KUKA KRL program: MyProgram_183().src

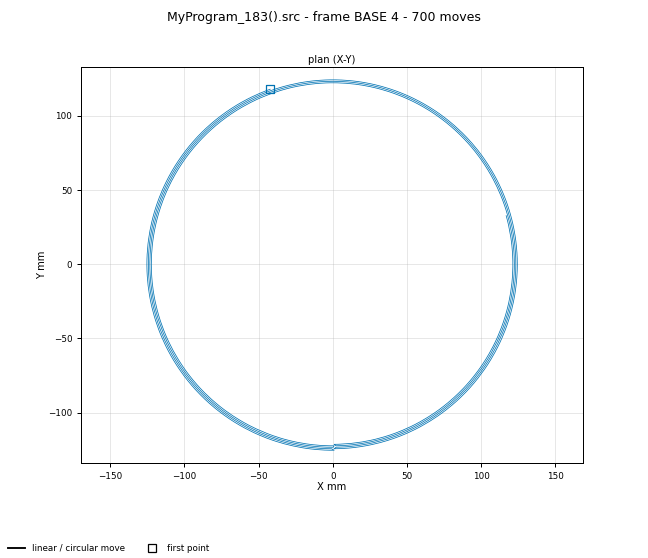
[picture p0: tool path of MyProgram_183().src in frame BASE 4, 700 of 700 moves have a stored position in this frame; points joined in program order, loops and branches not executed]
&ACCESS RVP
&REL 1
&PARAM TEMPLATE = C:\KRC\Roboter\Template\vorgabe
&PARAM EDITMASK = *
DEF MyProgram_183()
; ---- Setting reference (Base) ----
$BASE = BASE_DATA[4]

; --------------------------
; ---- Setting tool (TCP) ----
$TOOL = TOOL_DATA[3]
; --------------------------

$VEL.CP = VEL_APROX_PRINT
Startdeposition()
$VEL.CP = VEL_PRINT
LIN {X -42.2128,Y 118.0054,Z 134,A 105.9576,B 24.9444,C -1.7229,E1 24.9453,E2 340.2664} C_DIS
LIN {X -45.2291,Y 116.8823,Z 134,A 107.4306,B 24.9444,C -1.721,E1 24.9415,E2 338.7949} C_DIS
LIN {X -49.3483,Y 115.2042,Z 134,A 109.5085,B 24.9446,C -1.7201,E1 24.9361,E2 336.7143} C_DIS
LIN {X -52.4065,Y 113.845,Z 134,A 110.9287,B 24.945,C -1.7127,E1 24.9326,E2 335.3083} C_DIS
LIN {X -54.737,Y 112.7456,Z 134,A 112.3481,B 24.9444,C -1.722,E1 24.9289,E2 333.8631} C_DIS
LIN {X -57.7045,Y 111.2549,Z 134,A 113.8311,B 24.9447,C -1.7178,E1 24.9253,E2 332.3861} C_DIS
LIN {X -61.6733,Y 109.1057,Z 134,A 115.8056,B 24.9452,C -1.71,E1 24.9205,E2 330.4243} C_DIS
LIN {X -64.714,Y 107.3297,Z 134,A 117.5198,B 24.9451,C -1.7119,E1 24.9163,E2 328.7004} C_DIS
LIN {X -68.5088,Y 104.9484,Z 134,A 119.5092,B 24.9455,C -1.7052,E1 24.9117,E2 326.7206} C_DIS
LIN {X -71.9101,Y 102.6481,Z 134,A 121.4856,B 24.9455,C -1.706,E1 24.9071,E2 324.7356} C_DIS
LIN {X -75.2001,Y 100.2627,Z 134,A 123.3676,B 24.9456,C -1.7032,E1 24.9029,E2 322.8536} C_DIS
LIN {X -78.7307,Y 97.5142,Z 134,A 125.3322,B 24.9462,C -1.695,E1 24.8986,E2 320.9012} C_DIS
LIN {X -81.914,Y 94.856,Z 134,A 127.2839,B 24.9462,C -1.6933,E1 24.8944,E2 318.9461} C_DIS
LIN {X -85.115,Y 91.9953,Z 134,A 129.2878,B 24.9464,C -1.6905,E1 24.8903,E2 316.9406} C_DIS
LIN {X -88.2175,Y 89.0238,Z 134,A 131.2363,B 24.9468,C -1.6851,E1 24.8864,E2 314.997} C_DIS
LIN {X -91.0515,Y 86.1231,Z 134,A 133.1002,B 24.9471,C -1.6809,E1 24.8828,E2 313.1351} C_DIS
LIN {X -93.789,Y 83.1336,Z 134,A 134.9639,B 24.9473,C -1.6766,E1 24.8793,E2 311.2732} C_DIS
LIN {X -96.7243,Y 79.6996,Z 134,A 137.0122,B 24.9477,C -1.6704,E1 24.8757,E2 309.2303} C_DIS
LIN {X -99.3061,Y 76.4591,Z 134,A 138.9694,B 24.9479,C -1.6681,E1 24.8723,E2 307.2693} C_DIS
LIN {X -101.7154,Y 73.2235,Z 134,A 140.8408,B 24.9481,C -1.6643,E1 24.8692,E2 305.398} C_DIS
LIN {X -104.0135,Y 69.9207,Z 134,A 142.6859,B 24.9484,C -1.6593,E1 24.8663,E2 303.5555} C_DIS
LIN {X -106.3234,Y 66.3544,Z 134,A 144.6,B 24.9488,C -1.6525,E1 24.8634,E2 301.6481} C_DIS
LIN {X -108.4861,Y 62.7559,Z 134,A 146.4839,B 24.9493,C -1.6452,E1 24.8608,E2 299.7716} C_DIS
LIN {X -110.4801,Y 59.1752,Z 134,A 148.3446,B 24.9497,C -1.6391,E1 24.8583,E2 297.9157} C_DIS
LIN {X -112.2559,Y 55.7297,Z 134,A 150.1087,B 24.95,C -1.6334,E1 24.8561,E2 296.1557} C_DIS
LIN {X -113.6473,Y 52.834,Z 134,A 151.5899,B 24.9502,C -1.6295,E1 24.8543,E2 294.6757} C_DIS
LIN {X -114.9101,Y 50.0286,Z 134,A 152.9838,B 24.9505,C -1.6246,E1 24.8527,E2 293.2859} C_DIS
LIN {X -116.1361,Y 47.1124,Z 134,A 154.4266,B 24.9508,C -1.62,E1 24.8512,E2 291.8461} C_DIS
LIN {X -117.0936,Y 44.6855,Z 134,A 155.7763,B 24.9506,C -1.6233,E1 24.8498,E2 290.481} C_DIS
LIN {X -118.3112,Y 41.3481,Z 134,A 157.2703,B 24.9513,C -1.6123,E1 24.8485,E2 289.0046} C_DIS
LIN {X -119.2715,Y 38.4909,Z 134,A 158.6738,B 24.9515,C -1.6091,E1 24.8472,E2 287.6008} C_DIS
LIN {X -120.2509,Y 35.3108,Z 134,A 160.1325,B 24.9519,C -1.6014,E1 24.8461,E2 286.1519} C_DIS
LIN {X -121.2912,Y 31.5618,Z 134,A 162.127,B 24.9517,C -1.6054,E1 24.8446,E2 284.1364} C_DIS
LIN {X -122.0537,Y 28.467,Z 134,A 163.5459,B 24.9521,C -1.5989,E1 24.8437,E2 282.7246} C_DIS
LIN {X -122.7572,Y 25.2565,Z 134,A 164.9795,B 24.9526,C -1.591,E1 24.8429,E2 281.3015} C_DIS
LIN {X -123.2656,Y 22.6512,Z 134,A 166.2569,B 24.9526,C -1.5899,E1 24.8422,E2 280.0191} C_DIS
LIN {X -123.8062,Y 19.4749,Z 134,A 167.6166,B 24.9532,C -1.58,E1 24.8416,E2 278.6749} C_DIS
LIN {X -124.2273,Y 16.5782,Z 134,A 169.0665,B 24.9532,C -1.5806,E1 24.841,E2 277.2148} C_DIS
LIN {X -124.5803,Y 13.6749,Z 134,A 170.3322,B 24.9536,C -1.573,E1 24.8406,E2 275.9597} C_DIS
LIN {X -124.9891,Y 9.2159,Z 134,A 172.3518,B 24.9541,C -1.5651,E1 24.8402,E2 273.9469} C_DIS
LIN {X -125.1413,Y 6.87,Z 134,A 173.5919,B 24.9539,C -1.569,E1 24.84,E2 272.6901} C_DIS
LIN {X -125.2828,Y 3.3838,Z 134,A 175.1553,B 24.9543,C -1.5623,E1 24.8398,E2 271.1331} C_DIS
LIN {X -125.3282,Y -0.6113,Z 134,A 177.0633,B 24.9544,C -1.56,E1 24.8398,E2 269.2192} C_DIS
LIN {X -125.2421,Y -4.6552,Z 134,A 178.83,B 24.955,C -1.5502,E1 24.8399,E2 267.4651} C_DIS
LIN {X -125.0735,Y -7.9936,Z 134,A -179.497,B 24.9549,C -1.5518,E1 24.8402,E2 265.7783} C_DIS
LIN {X -124.7744,Y -11.772,Z 134,A -178.0165,B 24.9559,C -1.5348,E1 24.8406,E2 264.3294} C_DIS
LIN {X -124.4807,Y -14.5538,Z 134,A -176.5766,B 24.9557,C -1.5379,E1 24.841,E2 262.8734} C_DIS
LIN {X -124.086,Y -17.6024,Z 134,A -175.2591,B 24.9562,C -1.5294,E1 24.8415,E2 261.5683} C_DIS
LIN {X -123.6205,Y -20.6188,Z 134,A -173.8852,B 24.9565,C -1.524,E1 24.8421,E2 260.1991} C_DIS
LIN {X -122.8716,Y -24.6945,Z 134,A -171.8482,B 24.9565,C -1.5244,E1 24.8432,E2 258.1492} C_DIS
LIN {X -122.0036,Y -28.6837,Z 134,A -169.8902,B 24.9565,C -1.5226,E1 24.8444,E2 256.1838} C_DIS
LIN {X -121.1814,Y -31.9735,Z 134,A -168.6179,B 24.9576,C -1.5053,E1 24.8452,E2 254.9455} C_DIS
LIN {X -120.4925,Y -34.4857,Z 134,A -167.1064,B 24.9569,C -1.5161,E1 24.8464,E2 253.3995} C_DIS
LIN {X -119.479,Y -37.8414,Z 134,A -165.6096,B 24.9575,C -1.5064,E1 24.8476,E2 251.9173} C_DIS
LIN {X -118.4872,Y -40.8404,Z 134,A -164.2077,B 24.9578,C -1.5001,E1 24.8489,E2 250.5223} C_DIS
LIN {X -117.4756,Y -43.6657,Z 134,A -162.801,B 24.958,C -1.4975,E1 24.8502,E2 249.1137} C_DIS
LIN {X -116.5014,Y -46.2062,Z 134,A -161.5799,B 24.9583,C -1.4928,E1 24.8515,E2 247.8971} C_DIS
LIN {X -115.2168,Y -49.3193,Z 134,A -159.9549,B 24.9583,C -1.4922,E1 24.8532,E2 246.2646} C_DIS
LIN {X -113.8491,Y -52.3977,Z 134,A -158.5355,B 24.9588,C -1.4822,E1 24.8549,E2 244.8611} C_DIS
LIN {X -112.7456,Y -54.737,Z 134,A -157.1048,B 24.9584,C -1.4901,E1 24.8566,E2 243.4038} C_DIS
LIN {X -111.2809,Y -57.6551,Z 134,A -155.6229,B 24.9587,C -1.4854,E1 24.8585,E2 241.9251} C_DIS
LIN {X -109.093,Y -61.6959,Z 134,A -153.6286,B 24.9593,C -1.4748,E1 24.8612,E2 239.9458} C_DIS
LIN {X -107.3297,Y -64.714,Z 134,A -151.9247,B 24.9593,C -1.4753,E1 24.8636,E2 238.2318} C_DIS
LIN {X -104.937,Y -68.5264,Z 134,A -149.9496,B 24.9597,C -1.466,E1 24.8666,E2 236.2688} C_DIS
LIN {X -102.7847,Y -71.7138,Z 134,A -148.1115,B 24.9597,C -1.4652,E1 24.8695,E2 234.4236} C_DIS
LIN {X -100.283,Y -75.1732,Z 134,A -146.0743,B 24.9598,C -1.4642,E1 24.8729,E2 232.3788} C_DIS
LIN {X -97.8084,Y -78.3659,Z 134,A -144.28,B 24.9602,C -1.4573,E1 24.876,E2 230.5925} C_DIS
LIN {X -95.2021,Y -81.5121,Z 134,A -142.348,B 24.9602,C -1.4559,E1 24.8795,E2 228.655} C_DIS
LIN {X -92.3809,Y -84.6955,Z 134,A -140.4316,B 24.9606,C -1.4501,E1 24.883,E2 226.7438} C_DIS
LIN {X -89.3624,Y -87.8744,Z 134,A -138.4231,B 24.9608,C -1.4459,E1 24.8869,E2 224.7366} C_DIS
LIN {X -86.2984,Y -90.8861,Z 134,A -136.419,B 24.961,C -1.4436,E1 24.891,E2 222.7298} C_DIS
LIN {X -83.1336,Y -93.789,Z 134,A -134.4735,B 24.9612,C -1.4388,E1 24.895,E2 220.7879} C_DIS
LIN {X -79.7295,Y -96.6996,Z 134,A -132.4395,B 24.9615,C -1.4342,E1 24.8993,E2 218.757} C_DIS
LIN {X -76.4591,Y -99.3061,Z 134,A -130.4738,B 24.9615,C -1.4332,E1 24.9037,E2 216.7865} C_DIS
LIN {X -73.119,Y -101.7901,Z 134,A -128.5626,B 24.9617,C -1.4303,E1 24.908,E2 214.8755} C_DIS
LIN {X -69.4511,Y -104.327,Z 134,A -126.6149,B 24.9621,C -1.4226,E1 24.9124,E2 212.9395} C_DIS
LIN {X -66.3544,Y -106.3234,Z 134,A -124.8572,B 24.9621,C -1.4235,E1 24.9166,E2 211.1743} C_DIS
LIN {X -62.6309,Y -108.5585,Z 134,A -122.9402,B 24.9624,C -1.4173,E1 24.9212,E2 209.266} C_DIS
LIN {X -59.1752,Y -110.4801,Z 134,A -121.0908,B 24.9624,C -1.4168,E1 24.9257,E2 207.4125} C_DIS
LIN {X -55.7324,Y -112.2545,Z 134,A -119.3679,B 24.9626,C -1.4123,E1 24.93,E2 205.6957} C_DIS
LIN {X -53.315,Y -113.4249,Z 134,A -118.0043,B 24.9624,C -1.4173,E1 24.9335,E2 204.317} C_DIS
LIN {X -50.0286,Y -114.9101,Z 134,A -116.5037,B 24.9628,C -1.4084,E1 24.9373,E2 202.8339} C_DIS
LIN {X -47.0776,Y -116.1501,Z 134,A -115.0402,B 24.9629,C -1.4069,E1 24.9411,E2 201.3706} C_DIS
LIN {X -44.6855,Y -117.0936,Z 134,A -113.712,B 24.9626,C -1.413,E1 24.9446,E2 200.025} C_DIS
LIN {X -41.3481,Y -118.3112,Z 134,A -112.237,B 24.9631,C -1.4044,E1 24.9484,E2 198.5675} C_DIS
LIN {X -38.3419,Y -119.3191,Z 134,A -110.8033,B 24.9631,C -1.4025,E1 24.9522,E2 197.1356} C_DIS
LIN {X -35.3348,Y -120.2439,Z 134,A -109.3676,B 24.9632,C -1.4014,E1 24.956,E2 195.7002} C_DIS
LIN {X -32.5893,Y -121.0172,Z 134,A -108.2282,B 24.9637,C -1.3926,E1 24.9591,E2 194.58} C_DIS
LIN {X -29.5959,Y -121.7837,Z 134,A -106.7428,B 24.9635,C -1.3953,E1 24.9631,E2 193.086} C_DIS
LIN {X -26.6178,Y -122.469,Z 134,A -105.2134,B 24.9632,C -1.401,E1 24.9673,E2 191.5412} C_DIS
LIN {X -23.8287,Y -123.0424,Z 134,A -104.0673,B 24.9637,C -1.3929,E1 24.9704,E2 190.413} C_DIS
LIN {X -20.9206,Y -123.5701,Z 134,A -102.555,B 24.9633,C -1.4002,E1 24.9746,E2 188.8816} C_DIS
LIN {X -18.2655,Y -123.9913,Z 134,A -101.2825,B 24.9632,C -1.402,E1 24.9781,E2 187.6039} C_DIS
LIN {X -14.8953,Y -124.44,Z 134,A -99.7709,B 24.9633,C -1.3997,E1 24.9823,E2 186.0967} C_DIS
LIN {X -11.2615,Y -124.8234,Z 134,A -97.9671,B 24.963,C -1.406,E1 24.9874,E2 184.2769} C_DIS
LIN {X -7.9927,Y -125.0736,Z 134,A -96.7028,B 24.9636,C -1.3946,E1 24.9908,E2 183.0393} C_DIS
LIN {X -5.5873,Y -125.2058,Z 134,A -95.4107,B 24.9631,C -1.404,E1 24.9945,E2 181.7246} C_DIS
LIN {X -2.2482,Y -125.3084,Z 134,A -94.08,B 24.9636,C -1.3946,E1 24.9981,E2 180.416} C_DIS
LIN {X 0.8896,Y -125.3254,Z 134,A -92.9496,B 24.9643,C -1.38,E1 25.0012,E2 179.3201} C_DIS
Enddeposition()
LIN {X 0.8896,Y -125.3254,Z 134,A -92.9496,B 24.9643,C -1.38,E1 25.0012,E2 179.3201} C_DIS
Startdeposition()
$VEL.CP = VEL_PRINT
LIN {X -0.8291,Y -124.3295,Z 134,A -94.093,B 24.9643,C -1.3803,E1 24.998,E2 180.4627} C_DIS
LIN {X -4.7488,Y -124.2414,Z 134,A -95.8527,B 24.9643,C -1.3824,E1 24.9931,E2 182.2179} C_DIS
LIN {X -8.5607,Y -124.038,Z 134,A -97.7312,B 24.9645,C -1.3766,E1 24.9878,E2 184.1107} C_DIS
LIN {X -13.0048,Y -123.6503,Z 134,A -99.6905,B 24.9643,C -1.3814,E1 24.9824,E2 186.0598} C_DIS
LIN {X -16.1934,Y -123.2729,Z 134,A -101.1295,B 24.9641,C -1.3836,E1 24.9784,E2 187.4945} C_DIS
LIN {X -19.8425,Y -122.7399,Z 134,A -102.89,B 24.9643,C -1.3811,E1 24.9736,E2 189.2625} C_DIS
LIN {X -24.0406,Y -121.9876,Z 134,A -104.8827,B 24.9643,C -1.3805,E1 24.9681,E2 191.2585} C_DIS
LIN {X -27.1247,Y -121.3383,Z 134,A -106.231,B 24.964,C -1.3861,E1 24.9644,E2 192.5951} C_DIS
LIN {X -30.2211,Y -120.6036,Z 134,A -107.7557,B 24.9641,C -1.3842,E1 24.9603,E2 194.1265} C_DIS
LIN {X -34.3893,Y -119.4825,Z 134,A -109.7988,B 24.9641,C -1.383,E1 24.9548,E2 196.1758} C_DIS
LIN {X -41.2804,Y -117.2802,Z 134,A -113.1988,B 24.9641,C -1.3825,E1 24.9457,E2 199.5831} C_DIS
LIN {X -44.9084,Y -115.938,Z 134,A -114.9299,B 24.964,C -1.3867,E1 24.9412,E2 201.308} C_DIS
LIN {X -48.9847,Y -114.276,Z 134,A -117.101,B 24.9642,C -1.3822,E1 24.9356,E2 203.4948} C_DIS
LIN {X -53.007,Y -112.4679,Z 134,A -119.021,B 24.9638,C -1.3897,E1 24.9308,E2 205.4016} C_DIS
LIN {X -55.7905,Y -111.1136,Z 134,A -120.4058,B 24.9636,C -1.3934,E1 24.9273,E2 206.7812} C_DIS
LIN {X -58.7245,Y -109.5913,Z 134,A -121.9414,B 24.9636,C -1.3949,E1 24.9235,E2 208.3176} C_DIS
LIN {X -62.3051,Y -107.5959,Z 134,A -123.8517,B 24.9635,C -1.3966,E1 24.9189,E2 210.2295} C_DIS
LIN {X -66.3823,Y -105.1294,Z 134,A -126.041,B 24.9633,C -1.4002,E1 24.9137,E2 212.417} C_DIS
LIN {X -69.9315,Y -102.803,Z 134,A -128.0254,B 24.9632,C -1.4021,E1 24.9091,E2 214.4035} C_DIS
LIN {X -73.3696,Y -100.3782,Z 134,A -129.6623,B 24.9623,C -1.4193,E1 24.9054,E2 216.0052} C_DIS
LIN {X -75.9762,Y -98.4199,Z 134,A -131.4708,B 24.9629,C -1.408,E1 24.9013,E2 217.8471} C_DIS
LIN {X -79.2164,Y -95.8309,Z 134,A -133.4121,B 24.9627,C -1.4102,E1 24.8971,E2 219.7905} C_DIS
LIN {X -82.6197,Y -92.9134,Z 134,A -135.2958,B 24.9621,C -1.4226,E1 24.8932,E2 221.6521} C_DIS
LIN {X -85.1856,Y -90.5662,Z 134,A -137.0947,B 24.9624,C -1.417,E1 24.8895,E2 223.4716} C_DIS
LIN {X -88.264,Y -87.5686,Z 134,A -139.0924,B 24.9622,C -1.4204,E1 24.8855,E2 225.4696} C_DIS
LIN {X -91.3259,Y -84.371,Z 134,A -141.1608,B 24.962,C -1.4237,E1 24.8815,E2 227.5392} C_DIS
LIN {X -93.89,Y -81.5081,Z 134,A -142.9209,B 24.9618,C -1.4283,E1 24.8783,E2 229.2963} C_DIS
LIN {X -96.738,Y -78.106,Z 134,A -144.9464,B 24.9615,C -1.434,E1 24.8747,E2 231.3174} C_DIS
LIN {X -99.4141,Y -74.6707,Z 134,A -146.9963,B 24.9613,C -1.437,E1 24.8712,E2 233.37} C_DIS
LIN {X -101.9099,Y -71.2267,Z 134,A -148.9684,B 24.9611,C -1.4415,E1 24.868,E2 235.3412} C_DIS
LIN {X -103.9347,Y -68.2379,Z 134,A -150.697,B 24.961,C -1.4429,E1 24.8653,E2 237.075} C_DIS
LIN {X -106.3933,Y -64.3372,Z 134,A -152.7469,B 24.9605,C -1.4519,E1 24.8624,E2 239.1139} C_DIS
LIN {X -108.4732,Y -60.7651,Z 134,A -154.8338,B 24.9607,C -1.449,E1 24.8594,E2 241.2186} C_DIS
LIN {X -110.6976,Y -56.6076,Z 134,A -156.8123,B 24.9599,C -1.4638,E1 24.8569,E2 243.1725} C_DIS
LIN {X -112.4921,Y -52.9564,Z 134,A -158.9864,B 24.9603,C -1.4558,E1 24.8543,E2 245.3772} C_DIS
LIN {X -113.8392,Y -49.995,Z 134,A -160.2929,B 24.9596,C -1.4687,E1 24.8528,E2 246.6603} C_DIS
LIN {X -115.3156,Y -46.483,Z 134,A -161.9287,B 24.959,C -1.4792,E1 24.8511,E2 248.2801} C_DIS
LIN {X -116.7566,Y -42.739,Z 134,A -164.3001,B 24.96,C -1.4617,E1 24.8487,E2 250.7067} C_DIS
LIN {X -118.0857,Y -38.9141,Z 134,A -165.7588,B 24.9587,C -1.4853,E1 24.8475,E2 252.1175} C_DIS
LIN {X -119.2653,Y -35.1314,Z 134,A -167.3661,B 24.9578,C -1.5006,E1 24.8462,E2 253.6976} C_DIS
LIN {X -120.1074,Y -32.1344,Z 134,A -168.9132,B 24.9578,C -1.5001,E1 24.845,E2 255.255} C_DIS
LIN {X -120.8429,Y -29.2475,Z 134,A -170.3453,B 24.9578,C -1.5017,E1 24.8441,E2 256.6915} C_DIS
LIN {X -121.6967,Y -25.4715,Z 134,A -173.356,B 24.9604,C -1.4539,E1 24.8423,E2 259.8339} C_DIS
LIN {X -123.0108,Y -18.0842,Z 134,A -175.4738,B 24.9565,C -1.5233,E1 24.8414,E2 261.799} C_DIS
LIN {X -123.6979,Y -12.5594,Z 134,A -178.3129,B 24.9567,C -1.5195,E1 24.8405,E2 264.6641} C_DIS
LIN {X -124.1612,Y -6.522,Z 134,A 178.9873,B 24.956,C -1.5325,E1 24.84,E2 267.349} C_DIS
LIN {X -124.2881,Y -3.3114,Z 134,A 177.0622,B 24.9568,C -1.518,E1 24.8398,E2 269.3205} C_DIS
LIN {X -124.3322,Y 0.5419,Z 134,A 175.6181,B 24.9557,C -1.5382,E1 24.8398,E2 270.725} C_DIS
LIN {X -124.184,Y 6.0687,Z 134,A 173.0923,B 24.9551,C -1.5476,E1 24.84,E2 273.2436} C_DIS
LIN {X -123.9381,Y 9.9053,Z 134,A 171.2479,B 24.955,C -1.5502,E1 24.8404,E2 275.0929} C_DIS
LIN {X -123.5359,Y 14.0627,Z 134,A 169.433,B 24.9543,C -1.5613,E1 24.8409,E2 276.8922} C_DIS
LIN {X -123.093,Y 17.5083,Z 134,A 167.7056,B 24.9543,C -1.561,E1 24.8416,E2 278.6306} C_DIS
LIN {X -122.5787,Y 20.809,Z 134,A 165.4846,B 24.9558,C -1.5364,E1 24.8427,E2 280.9235} C_DIS
LIN {X -121.5645,Y 26.0864,Z 134,A 163.7741,B 24.9534,C -1.5778,E1 24.8436,E2 282.5454} C_DIS
LIN {X -120.8639,Y 29.1601,Z 134,A 162.3759,B 24.9529,C -1.5849,E1 24.8445,E2 283.935} C_DIS
LIN {X -120.0864,Y 32.2132,Z 134,A 160.7926,B 24.953,C -1.5838,E1 24.8456,E2 285.5301} C_DIS
LIN {X -118.9565,Y 36.1635,Z 134,A 158.9999,B 24.9524,C -1.5942,E1 24.847,E2 287.3082} C_DIS
LIN {X -117.9617,Y 39.2863,Z 134,A 157.4009,B 24.9524,C -1.5951,E1 24.8484,E2 288.9142} C_DIS
LIN {X -116.6741,Y 42.965,Z 134,A 155.6314,B 24.9519,C -1.6019,E1 24.85,E2 290.6775} C_DIS
LIN {X -115.3326,Y 46.4408,Z 134,A 153.9134,B 24.9516,C -1.6073,E1 24.8518,E2 292.3924} C_DIS
LIN {X -114.2119,Y 49.133,Z 134,A 152.5,B 24.9516,C -1.6084,E1 24.8533,E2 293.8111} C_DIS
LIN {X -112.8301,Y 52.2275,Z 134,A 151.0165,B 24.951,C -1.6166,E1 24.855,E2 295.283} C_DIS
LIN {X -111.1514,Y 55.7163,Z 134,A 149.0903,B 24.951,C -1.6157,E1 24.8574,E2 297.2217} C_DIS
LIN {X -109.5282,Y 58.842,Z 134,A 147.4976,B 24.9507,C -1.6219,E1 24.8595,E2 298.8081} C_DIS
LIN {X -107.5727,Y 62.3452,Z 134,A 145.6296,B 24.9504,C -1.6265,E1 24.862,E2 300.6749} C_DIS
LIN {X -105.3698,Y 66.001,Z 134,A 143.5621,B 24.9504,C -1.6278,E1 24.8651,E2 302.75} C_DIS
LIN {X -102.9906,Y 69.6545,Z 134,A 141.5508,B 24.95,C -1.6334,E1 24.8682,E2 304.758} C_DIS
LIN {X -100.4113,Y 73.3246,Z 134,A 139.4495,B 24.9497,C -1.6377,E1 24.8716,E2 306.8594} C_DIS
LIN {X -97.72,Y 76.874,Z 134,A 137.431,B 24.9493,C -1.6447,E1 24.875,E2 308.8707} C_DIS
LIN {X -94.9868,Y 80.2276,Z 134,A 135.3766,B 24.9491,C -1.6473,E1 24.8787,E2 310.9284} C_DIS
LIN {X -92.0924,Y 83.5332,Z 134,A 133.4305,B 24.9486,C -1.6561,E1 24.8823,E2 312.8624} C_DIS
LIN {X -89.2646,Y 86.5484,Z 134,A 131.4611,B 24.9485,C -1.658,E1 24.8861,E2 314.8358} C_DIS
LIN {X -86.162,Y 89.6383,Z 134,A 129.4066,B 24.9483,C -1.6612,E1 24.8902,E2 316.8911} C_DIS
LIN {X -83.1514,Y 92.4376,Z 134,A 127.519,B 24.948,C -1.666,E1 24.8941,E2 318.775} C_DIS
LIN {X -79.9464,Y 95.2227,Z 134,A 125.6039,B 24.9476,C -1.6723,E1 24.8981,E2 320.6824} C_DIS
LIN {X -76.572,Y 97.9572,Z 134,A 123.5711,B 24.9474,C -1.6753,E1 24.9026,E2 322.7157} C_DIS
LIN {X -73.3404,Y 100.3997,Z 134,A 121.695,B 24.9472,C -1.6788,E1 24.9068,E2 324.5901} C_DIS
LIN {X -70.114,Y 102.6787,Z 134,A 119.8614,B 24.947,C -1.6819,E1 24.911,E2 326.4226} C_DIS
LIN {X -66.6424,Y 104.9653,Z 134,A 117.9034,B 24.9469,C -1.6838,E1 24.9156,E2 328.3826} C_DIS
LIN {X -62.7596,Y 107.3317,Z 134,A 115.8441,B 24.9465,C -1.6893,E1 24.9205,E2 330.4351} C_DIS
LIN {X -59.0643,Y 109.4088,Z 134,A 113.8454,B 24.9465,C -1.6907,E1 24.9254,E2 332.4362} C_DIS
LIN {X -55.2264,Y 111.3932,Z 134,A 112.2081,B 24.9452,C -1.7101,E1 24.9293,E2 334.0319} C_DIS
LIN {X -51.4492,Y 113.1896,Z 134,A 109.8903,B 24.9461,C -1.6953,E1 24.9353,E2 336.3906} C_DIS
LIN {X -48.0206,Y 114.6839,Z 134,A 108.2868,B 24.9456,C -1.7033,E1 24.9394,E2 337.9787} C_DIS
LIN {X -45.2872,Y 115.7908,Z 134,A 106.3065,B 24.9473,C -1.677,E1 24.9447,E2 340.0259} C_DIS
LIN {X -40.8805,Y 117.4189,Z 134,A 104.7604,B 24.9453,C -1.7079,E1 24.9486,E2 341.5017} C_DIS
LIN {X -37.7579,Y 118.4598,Z 134,A 103.1894,B 24.9453,C -1.7072,E1 24.9528,E2 343.0771} C_DIS
LIN {X -33.5588,Y 119.7172,Z 134,A 100.6802,B 24.9467,C -1.687,E1 24.9597,E2 345.6382} C_DIS
LIN {X -29.4074,Y 120.8043,Z 134,A 99.4701,B 24.9443,C -1.7242,E1 24.9627,E2 346.7617} C_DIS
LIN {X -22.7276,Y 122.2386,Z 134,A 96.0433,B 24.9449,C -1.714,E1 24.9722,E2 350.217} C_DIS
LIN {X -20.3015,Y 122.6634,Z 134,A 94.6081,B 24.9458,C -1.7009,E1 24.9762,E2 351.6844} C_DIS
LIN {X -16.898,Y 123.1803,Z 134,A 93.2781,B 24.945,C -1.7138,E1 24.9798,E2 352.985} C_DIS
LIN {X -13.0642,Y 123.644,Z 134,A 91.5095,B 24.9449,C -1.7153,E1 24.9847,E2 354.751} C_DIS
LIN {X -9.0218,Y 124.0043,Z 134,A 89.6198,B 24.9449,C -1.7153,E1 24.9899,E2 356.6416} C_DIS
LIN {X -5.171,Y 124.2249,Z 134,A 87.9265,B 24.9446,C -1.7199,E1 24.9946,E2 358.3246} C_DIS
LIN {X -1.7803,Y 124.3197,Z 134,A 86.3238,B 24.9446,C -1.7184,E1 24.9991,E2 359.9309} C_DIS
LIN {X 1.8786,Y 124.3181,Z 134,A 84.5937,B 24.9448,C -1.7166,E1 25.004,E2 361.6651} C_DIS
LIN {X 5.9235,Y 124.1913,Z 134,A 82.6719,B 24.9449,C -1.7141,E1 25.0093,E2 363.5923} C_DIS
LIN {X 10.0163,Y 123.9287,Z 134,A 80.9026,B 24.9446,C -1.7197,E1 25.0142,E2 365.3476} C_DIS
LIN {X 13.2988,Y 123.6187,Z 134,A 79.3791,B 24.9446,C -1.7193,E1 25.0185,E2 366.8709} C_DIS
LIN {X 16.8352,Y 123.1888,Z 134,A 77.8073,B 24.9444,C -1.7222,E1 25.0228,E2 368.4346} C_DIS
LIN {X 20.7641,Y 122.5862,Z 134,A 75.8052,B 24.945,C -1.7136,E1 25.0284,E2 370.4553} C_DIS
LIN {X 24.909,Y 121.8112,Z 134,A 73.9642,B 24.9447,C -1.7176,E1 25.0334,E2 372.2845} C_DIS
LIN {X 28.1891,Y 121.0952,Z 134,A 72.2621,B 24.9452,C -1.7094,E1 25.0381,E2 374.0038} C_DIS
LIN {X 32.8459,Y 119.9166,Z 134,A 70.304,B 24.9445,C -1.7202,E1 25.0433,E2 375.9333} C_DIS
LIN {X 38.4183,Y 118.2488,Z 134,A 67.4575,B 24.9452,C -1.7101,E1 25.0509,E2 378.7985} C_DIS
LIN {X 42.0457,Y 117.0066,Z 134,A 65.7953,B 24.945,C -1.7136,E1 25.0553,E2 380.4491} C_DIS
LIN {X 44.879,Y 115.9494,Z 134,A 64.5599,B 24.9446,C -1.7199,E1 25.0584,E2 381.667} C_DIS
LIN {X 48.497,Y 114.4849,Z 134,A 62.5282,B 24.9454,C -1.7066,E1 25.0638,E2 383.7253} C_DIS
LIN {X 51.4448,Y 113.1916,Z 134,A 61.0841,B 24.9454,C -1.7068,E1 25.0674,E2 385.1654} C_DIS
LIN {X 54.3981,Y 111.8018,Z 134,A 59.4753,B 24.9458,C -1.6999,E1 25.0715,E2 386.7864} C_DIS
LIN {X 58.6019,Y 109.6572,Z 134,A 57.3728,B 24.9458,C -1.7005,E1 25.0767,E2 388.8817} C_DIS
LIN {X 61.5153,Y 108.0494,Z 134,A 55.8274,B 24.946,C -1.6977,E1 25.0805,E2 390.429} C_DIS
LIN {X 65.3025,Y 105.8041,Z 134,A 53.8059,B 24.9462,C -1.6949,E1 25.0853,E2 392.4507} C_DIS
LIN {X 68.8681,Y 103.5182,Z 134,A 51.876,B 24.9462,C -1.6929,E1 25.0898,E2 394.3792} C_DIS
LIN {X 71.727,Y 101.5581,Z 134,A 50.2654,B 24.9465,C -1.6895,E1 25.0935,E2 395.9922} C_DIS
LIN {X 75.2073,Y 99.0092,Z 134,A 48.3095,B 24.9466,C -1.6875,E1 25.0979,E2 397.9459} C_DIS
LIN {X 78.4367,Y 96.4706,Z 134,A 46.239,B 24.9474,C -1.6751,E1 25.1024,E2 400.0378} C_DIS
LIN {X 81.8563,Y 93.5861,Z 134,A 43.2776,B 24.9504,C -1.6271,E1 25.1089,E2 403.1009} C_DIS
LIN {X 87.2524,Y 88.577,Z 134,A 40.9535,B 24.9476,C -1.6722,E1 25.1133,E2 405.3089} C_DIS
LIN {X 90.2407,Y 85.5307,Z 134,A 39.0371,B 24.9477,C -1.6703,E1 25.117,E2 407.2215} C_DIS
LIN {X 93.8684,Y 81.5328,Z 134,A 35.6978,B 24.9507,C -1.6225,E1 25.1233,E2 410.6587} C_DIS
LIN {X 97.8335,Y 76.7294,Z 134,A 33.7029,B 24.9484,C -1.6588,E1 25.1267,E2 412.5586} C_DIS
LIN {X 100.4155,Y 73.3188,Z 134,A 32.0034,B 24.9479,C -1.6674,E1 25.1294,E2 414.2295} C_DIS
LIN {X 102.1863,Y 70.8295,Z 134,A 30.3373,B 24.9489,C -1.6509,E1 25.1322,E2 415.9265} C_DIS
LIN {X 104.5096,Y 67.355,Z 134,A 28.3744,B 24.9494,C -1.6439,E1 25.1352,E2 417.8959} C_DIS
LIN {X 106.8778,Y 63.5292,Z 134,A 26.3523,B 24.9495,C -1.6409,E1 25.1381,E2 419.9149} C_DIS
LIN {X 109.0073,Y 59.8022,Z 134,A 24.5598,B 24.9493,C -1.6448,E1 25.1405,E2 421.6888} C_DIS
LIN {X 110.6401,Y 56.7207,Z 134,A 22.9832,B 24.9495,C -1.6419,E1 25.1426,E2 423.264} C_DIS
LIN {X 112.0561,Y 53.8689,Z 134,A 21.3973,B 24.9501,C -1.6317,E1 25.1445,E2 424.8655} C_DIS
LIN {X 113.5493,Y 50.6452,Z 134,A 19.76,B 24.9504,C -1.6269,E1 25.1464,E2 426.5051} C_DIS
LIN {X 114.9681,Y 47.34,Z 134,A 18.0406,B 24.9509,C -1.6189,E1 25.1483,E2 428.234} C_DIS
LIN {X 116.3029,Y 43.9561,Z 134,A 16.4624,B 24.9509,C -1.6189,E1 25.1499,E2 429.8035} C_DIS
LIN {X 117.4019,Y 40.9294,Z 134,A 14.9876,B 24.9511,C -1.6149,E1 25.1513,E2 431.2795} C_DIS
LIN {X 118.6726,Y 37.0909,Z 134,A 12.7365,B 24.9527,C -1.5895,E1 25.1532,E2 433.5777} C_DIS
LIN {X 119.6887,Y 33.6607,Z 134,A 11.4992,B 24.9517,C -1.6052,E1 25.1541,E2 434.7707} C_DIS
LIN {X 120.6461,Y 30.0536,Z 134,A 9.6892,B 24.9523,C -1.5953,E1 25.1554,E2 436.5938} C_DIS
LIN {X 121.32,Y 27.205,Z 134,A 8.2489,B 24.9528,C -1.5864,E1 25.1563,E2 438.0467} C_DIS
LIN {X 122.0732,Y 23.5927,Z 134,A 6.6098,B 24.953,C -1.5841,E1 25.1572,E2 439.6816} C_DIS
LIN {X 122.8174,Y 19.35,Z 134,A 4.7647,B 24.953,C -1.5848,E1 25.158,E2 441.5142} C_DIS
LIN {X 123.3382,Y 15.695,Z 134,A 3.1294,B 24.953,C -1.5827,E1 25.1586,E2 443.1449} C_DIS
LIN {X 123.7731,Y 11.7765,Z 134,A 1.2177,B 24.9537,C -1.572,E1 25.1592,E2 445.0705} C_DIS
LIN {X 124.0952,Y 7.6714,Z 134,A -0.5805,B 24.9537,C -1.5709,E1 25.1595,E2 446.8606} C_DIS
LIN {X 124.2634,Y 4.1838,Z 134,A -2.3622,B 24.9546,C -1.5568,E1 25.1597,E2 448.6649} C_DIS
LIN {X 124.3326,Y -0.4646,Z 134,A -4.3597,B 24.9546,C -1.5571,E1 25.1597,E2 450.6497} C_DIS
LIN {X 124.2505,Y -4.5163,Z 134,A -6.2337,B 24.9549,C -1.5507,E1 25.1597,E2 452.5278} C_DIS
LIN {X 124.0221,Y -8.7778,Z 134,A -8.1363,B 24.9551,C -1.5475,E1 25.1593,E2 454.4266} C_DIS
LIN {X 123.6914,Y -12.6229,Z 134,A -10.1576,B 24.9562,C -1.5292,E1 25.1588,E2 456.479} C_DIS
LIN {X 123.1034,Y -17.4361,Z 134,A -12.1141,B 24.9558,C -1.5361,E1 25.1581,E2 458.4078} C_DIS
LIN {X 122.5568,Y -20.9404,Z 134,A -13.699,B 24.956,C -1.5333,E1 25.1573,E2 459.99} C_DIS
LIN {X 121.7403,Y -25.2573,Z 134,A -15.8465,B 24.9567,C -1.5204,E1 25.1562,E2 462.1554} C_DIS
LIN {X 120.5423,Y -30.4627,Z 134,A -18.1622,B 24.9567,C -1.5198,E1 25.1547,E2 464.4589} C_DIS
LIN {X 119.5443,Y -34.1771,Z 134,A -20.035,B 24.9573,C -1.509,E1 25.1533,E2 466.3465} C_DIS
LIN {X 118.4673,Y -37.7343,Z 134,A -22.1037,B 24.9587,C -1.4854,E1 25.1515,E2 468.459} C_DIS
LIN {X 117.1683,Y -41.5973,Z 134,A -23.5676,B 24.9578,C -1.5005,E1 25.1502,E2 469.8792} C_DIS
LIN {X 116.029,Y -44.6742,Z 134,A -25.0458,B 24.958,C -1.4975,E1 25.1487,E2 471.3562} C_DIS
LIN {X 114.1384,Y -49.303,Z 134,A -27.3023,B 24.9583,C -1.4927,E1 25.1463,E2 473.6115} C_DIS
LIN {X 112.6911,Y -52.5282,Z 134,A -29.0277,B 24.9588,C -1.4828,E1 25.1443,E2 475.3509} C_DIS
LIN {X 110.9836,Y -56.046,Z 134,A -30.6424,B 24.9586,C -1.4868,E1 25.1423,E2 476.9475} C_DIS
LIN {X 109.2985,Y -59.2683,Z 134,A -32.6734,B 24.9599,C -1.4637,E1 25.1396,E2 479.0224} C_DIS
LIN {X 106.5966,Y -64.0009,Z 134,A -34.9749,B 24.9597,C -1.467,E1 25.1364,E2 481.3043} C_DIS
LIN {X 104.3155,Y -67.6541,Z 134,A -36.8626,B 24.9597,C -1.4662,E1 25.1335,E2 483.1844} C_DIS
LIN {X 102.073,Y -70.9923,Z 134,A -38.7466,B 24.9601,C -1.4593,E1 25.1306,E2 485.0752} C_DIS
LIN {X 97.8398,Y -76.7215,Z 134,A -41.9982,B 24.9605,C -1.4518,E1 25.1251,E2 488.329} C_DIS
LIN {X 95.2544,Y -79.9087,Z 134,A -43.8935,B 24.9608,C -1.4466,E1 25.1217,E2 490.2279} C_DIS
LIN {X 92.4664,Y -83.1192,Z 134,A -45.5836,B 24.9603,C -1.4551,E1 25.1187,E2 491.8903} C_DIS
LIN {X 89.3547,Y -86.4554,Z 134,A -48.0777,B 24.9617,C -1.4299,E1 25.1138,E2 494.433} C_DIS
LIN {X 85.8133,Y -89.9716,Z 134,A -50.1803,B 24.9615,C -1.4342,E1 25.1096,E2 496.5167} C_DIS
LIN {X 82.7989,Y -92.7533,Z 134,A -51.8323,B 24.9611,C -1.4417,E1 25.1063,E2 498.1443} C_DIS
LIN {X 80.5677,Y -94.6976,Z 134,A -53.6518,B 24.9625,C -1.4156,E1 25.1023,E2 500.0182} C_DIS
LIN {X 76.4712,Y -98.0362,Z 134,A -55.929,B 24.9623,C -1.4181,E1 25.0974,E2 502.2811} C_DIS
LIN {X 73.0548,Y -100.6072,Z 134,A -57.6985,B 24.962,C -1.424,E1 25.0935,E2 504.0303} C_DIS
LIN {X 70.8619,Y -102.1637,Z 134,A -58.9427,B 24.9622,C -1.4211,E1 25.0906,E2 505.277} C_DIS
LIN {X 67.5129,Y -104.4072,Z 134,A -60.7343,B 24.9622,C -1.4207,E1 25.0864,E2 507.0636} C_DIS
LIN {X 65.5653,Y -105.641,Z 134,A -63.1333,B 24.9657,C -1.3526,E1 25.0804,E2 509.6159} C_DIS
LIN {X 58.9676,Y -109.4607,Z 134,A -65.4755,B 24.9631,C -1.4039,E1 25.075,E2 511.8302} C_DIS
LIN {X 55.4689,Y -111.2736,Z 134,A -67.4653,B 24.9637,C -1.3922,E1 25.0699,E2 513.8421} C_DIS
LIN {X 50.9713,Y -113.4034,Z 134,A -69.5424,B 24.9633,C -1.3993,E1 25.0647,E2 515.8972} C_DIS
LIN {X 47.9188,Y -114.7264,Z 134,A -71.0193,B 24.9633,C -1.3998,E1 25.0609,E2 517.3695} C_DIS
LIN {X 44.7924,Y -115.9831,Z 134,A -72.6284,B 24.9636,C -1.3948,E1 25.0567,E2 518.9868} C_DIS
LIN {X 40.8931,Y -117.4145,Z 134,A -74.5959,B 24.9638,C -1.3896,E1 25.0515,E2 520.9625} C_DIS
LIN {X 36.7266,Y -118.7841,Z 134,A -76.5273,B 24.9638,C -1.3916,E1 25.0464,E2 522.8857} C_DIS
LIN {X 32.0614,Y -120.1269,Z 134,A -78.7111,B 24.9638,C -1.3916,E1 25.0406,E2 525.0656} C_DIS
LIN {X 29.0285,Y -120.8957,Z 134,A -80.1095,B 24.9637,C -1.3923,E1 25.0368,E2 526.4604} C_DIS
LIN {X 26.2861,Y -121.5214,Z 134,A -81.4472,B 24.9639,C -1.3891,E1 25.0331,E2 527.804} C_DIS
LIN {X 23.117,Y -122.1641,Z 134,A -82.8879,B 24.9638,C -1.3902,E1 25.0292,E2 529.2403} C_DIS
LIN {X 19.0916,Y -122.8574,Z 134,A -84.8849,B 24.9642,C -1.3832,E1 25.0237,E2 531.2519} C_DIS
LIN {X 14.4737,Y -123.4869,Z 134,A -87.0325,B 24.9642,C -1.3818,E1 25.0177,E2 533.401} C_DIS
LIN {X 10.5811,Y -123.881,Z 134,A -88.8496,B 24.9643,C -1.3802,E1 25.0126,E2 535.221} C_DIS
LIN {X 5.5584,Y -124.2097,Z 134,A -91.2605,B 24.9646,C -1.3748,E1 25.0059,E2 537.6437} C_DIS
LIN {X 0.8889,Y -124.3282,Z 134,A -93.2314,B 24.9642,C -1.3829,E1 25.0004,E2 539.5951} C_DIS
Enddeposition()
LIN {X 0.8889,Y -124.3282,Z 134,A -93.2314,B 24.9642,C -1.3829,E1 25.0004,E2 539.5951} C_DIS
Startdeposition()
$VEL.CP = VEL_PRINT
LIN {X 2.1717,Y -123.3168,Z 134,A -91.8897,B 24.9613,C -1.4365,E1 25.0045,E2 538.1265} C_DIS
LIN {X 8.2446,Y -123.0617,Z 134,A -89.0343,B 24.9613,C -1.4391,E1 25.0125,E2 535.2658} C_DIS
LIN {X 12.0717,Y -122.7439,Z 134,A -87.4105,B 24.9616,C -1.4323,E1 25.017,E2 533.6593} C_DIS
LIN {X 17.5172,Y -122.0854,Z 134,A -84.8105,B 24.9613,C -1.4365,E1 25.0242,E2 531.0514} C_DIS
LIN {X 24.3404,Y -120.9102,Z 134,A -81.8727,B 24.9619,C -1.4254,E1 25.0322,E2 528.1431} C_DIS
LIN {X 27.2234,Y -120.2938,Z 134,A -80.2489,B 24.9612,C -1.4391,E1 25.0367,E2 526.4889} C_DIS
LIN {X 35.0315,Y -118.2564,Z 134,A -76.6036,B 24.9612,C -1.4379,E1 25.0465,E2 522.8521} C_DIS
LIN {X 37.8367,Y -117.3887,Z 134,A -75.0889,B 24.9608,C -1.447,E1 25.0506,E2 521.3187} C_DIS
LIN {X 42.839,Y -115.6574,Z 134,A -72.824,B 24.9611,C -1.4406,E1 25.0565,E2 519.0736} C_DIS
LIN {X 45.9897,Y -114.4403,Z 134,A -71.1203,B 24.9606,C -1.4495,E1 25.061,E2 517.3526} C_DIS
LIN {X 49.4131,Y -113.0053,Z 134,A -69.3767,B 24.9604,C -1.4531,E1 25.0655,E2 515.6047} C_DIS
LIN {X 55.4672,Y -110.1602,Z 134,A -66.4506,B 24.9607,C -1.4491,E1 25.0728,E2 512.6958} C_DIS
LIN {X 58.8738,Y -108.3789,Z 134,A -64.2684,B 24.9594,C -1.472,E1 25.0783,E2 510.4656} C_DIS
LIN {X 64.8049,Y -104.9405,Z 134,A -61.5752,B 24.9604,C -1.4533,E1 25.0847,E2 507.8249} C_DIS
LIN {X 68.7947,Y -102.3694,Z 134,A -58.7539,B 24.9585,C -1.4887,E1 25.0914,E2 504.9294} C_DIS
LIN {X 71.8369,Y -100.2573,Z 134,A -56.7634,B 24.9575,C -1.506,E1 25.096,E2 502.9048} C_DIS
LIN {X 75.9182,Y -97.2038,Z 134,A -55.3189,B 24.9598,C -1.4644,E1 25.099,E2 501.5639} C_DIS
LIN {X 80.6675,Y -93.2998,Z 134,A -51.6228,B 24.9571,C -1.5135,E1 25.1071,E2 497.7661} C_DIS
LIN {X 84.2327,Y -90.0942,Z 134,A -49.965,B 24.9584,C -1.4898,E1 25.1103,E2 496.171} C_DIS
LIN {X 89.5177,Y -84.8452,Z 134,A -46.4532,B 24.9578,C -1.501,E1 25.1173,E2 492.6477} C_DIS
LIN {X 93.5324,Y -80.3974,Z 134,A -44.0479,B 24.9585,C -1.489,E1 25.1217,E2 490.2815} C_DIS
LIN {X 95.7261,Y -77.7729,Z 134,A -41.6137,B 24.9558,C -1.5365,E1 25.1261,E2 487.7466} C_DIS
LIN {X 98.6826,Y -73.9855,Z 134,A -40.0717,B 24.9574,C -1.5072,E1 25.1286,E2 486.281} C_DIS
LIN {X 100.2936,Y -71.7862,Z 134,A -38.6736,B 24.9569,C -1.5175,E1 25.1309,E2 484.8654} C_DIS
LIN {X 102.6112,Y -68.4324,Z 134,A -36.8286,B 24.9567,C -1.5204,E1 25.1338,E2 483.0227} C_DIS
LIN {X 104.9424,Y -64.8018,Z 134,A -34.7777,B 24.9562,C -1.5286,E1 25.1369,E2 480.9629} C_DIS
LIN {X 107.2757,Y -60.861,Z 134,A -32.684,B 24.956,C -1.5331,E1 25.1398,E2 478.8692} C_DIS
LIN {X 110.0119,Y -55.7586,Z 134,A -30.1737,B 24.956,C -1.532,E1 25.143,E2 476.3747} C_DIS
LIN {X 111.4349,Y -52.8581,Z 134,A -28.625,B 24.9556,C -1.5391,E1 25.1449,E2 474.8177} C_DIS
LIN {X 114.3395,Y -46.2396,Z 134,A -25.5841,B 24.956,C -1.5332,E1 25.1483,E2 471.8073} C_DIS
LIN {X 115.6471,Y -42.8666,Z 134,A -23.5371,B 24.9546,C -1.5573,E1 25.1504,E2 469.715} C_DIS
LIN {X 117.0646,Y -38.8268,Z 134,A -20.7081,B 24.9516,C -1.6071,E1 25.153,E2 466.7845} C_DIS
LIN {X 118.881,Y -32.8497,Z 134,A -18.8452,B 24.9543,C -1.5626,E1 25.1543,E2 465.0371} C_DIS
LIN {X 120.4612,Y -26.4756,Z 134,A -15.8939,B 24.954,C -1.5673,E1 25.1562,E2 462.0918} C_DIS
LIN {X 121.502,Y -21.1947,Z 134,A -13.3224,B 24.9533,C -1.5791,E1 25.1576,E2 459.5076} C_DIS
LIN {X 121.9352,Y -18.5363,Z 134,A -11.9447,B 24.9526,C -1.5897,E1 25.1582,E2 458.113} C_DIS
LIN {X 122.8154,Y -11.3266,Z 134,A -8.7854,B 24.9526,C -1.5897,E1 25.1592,E2 454.9724} C_DIS
LIN {X 123.0264,Y -8.733,Z 134,A -7.4079,B 24.9519,C -1.6023,E1 25.1595,E2 453.5733} C_DIS
LIN {X 123.2515,Y -4.5653,Z 134,A -5.4294,B 24.9514,C -1.6107,E1 25.1597,E2 451.5867} C_DIS
LIN {X 123.3371,Y -0.305,Z 134,A -3.423,B 24.9509,C -1.6186,E1 25.1597,E2 449.5738} C_DIS
LIN {X 123.2657,Y 4.2006,Z 134,A -1.5618,B 24.9512,C -1.6135,E1 25.1597,E2 447.7355} C_DIS
LIN {X 123.1105,Y 7.4528,Z 134,A 0.0378,B 24.9506,C -1.623,E1 25.1594,E2 446.1233} C_DIS
LIN {X 122.7392,Y 12.1198,Z 134,A 2.4599,B 24.9494,C -1.6427,E1 25.1588,E2 443.6689} C_DIS
LIN {X 122.2097,Y 16.6387,Z 134,A 4.3878,B 24.9496,C -1.64,E1 25.1581,E2 441.7588} C_DIS
LIN {X 121.6068,Y 20.5803,Z 134,A 6.5689,B 24.9482,C -1.6628,E1 25.1571,E2 439.5367} C_DIS
LIN {X 120.9021,Y 24.3802,Z 134,A 7.8059,B 24.9496,C -1.6399,E1 25.1565,E2 438.361} C_DIS
LIN {X 120.2856,Y 27.2592,Z 134,A 9.5187,B 24.9482,C -1.6619,E1 25.1554,E2 436.6064} C_DIS
LIN {X 119.3803,Y 30.991,Z 134,A 11.1013,B 24.9485,C -1.6571,E1 25.1543,E2 435.0441} C_DIS
LIN {X 117.6831,Y 36.9153,Z 134,A 13.9516,B 24.948,C -1.6653,E1 25.1521,E2 432.1908} C_DIS
LIN {X 116.5629,Y 40.3079,Z 134,A 15.5215,B 24.948,C -1.6658,E1 25.1507,E2 430.6286} C_DIS
LIN {X 115.3887,Y 43.5565,Z 134,A 17.0955,B 24.9478,C -1.669,E1 25.1492,E2 429.0557} C_DIS
LIN {X 114.3835,Y 46.1304,Z 134,A 18.3583,B 24.9476,C -1.6718,E1 25.1478,E2 427.7935} C_DIS
LIN {X 113.1189,Y 49.1505,Z 134,A 19.9304,B 24.9472,C -1.6788,E1 25.1461,E2 426.2133} C_DIS
LIN {X 111.6416,Y 52.424,Z 134,A 21.7376,B 24.9464,C -1.6907,E1 25.144,E2 424.3879} C_DIS
LIN {X 108.8941,Y 57.9144,Z 134,A 24.3363,B 24.9467,C -1.6859,E1 25.1407,E2 421.8143} C_DIS
LIN {X 107.272,Y 60.8675,Z 134,A 25.9782,B 24.9462,C -1.6941,E1 25.1385,E2 420.1617} C_DIS
LIN {X 105.4781,Y 63.9253,Z 134,A 27.6621,B 24.9458,C -1.7004,E1 25.136,E2 418.4715} C_DIS
LIN {X 103.3021,Y 67.3855,Z 134,A 29.5828,B 24.9454,C -1.7065,E1 25.1331,E2 416.5459} C_DIS
LIN {X 100.0442,Y 72.1339,Z 134,A 32.0353,B 24.9457,C -1.7022,E1 25.1293,E2 414.1157} C_DIS
LIN {X 98.1148,Y 74.7368,Z 134,A 33.6919,B 24.945,C -1.7136,E1 25.1264,E2 412.4401} C_DIS
LIN {X 95.2144,Y 78.3978,Z 134,A 35.9604,B 24.9443,C -1.7238,E1 25.1224,E2 410.1582} C_DIS
LIN {X 92.4629,Y 81.6252,Z 134,A 37.8678,B 24.9443,C -1.7252,E1 25.119,E2 408.2559} C_DIS
LIN {X 89.4856,Y 84.8792,Z 134,A 39.8939,B 24.944,C -1.7287,E1 25.1151,E2 406.2304} C_DIS
LIN {X 86.5305,Y 87.8895,Z 134,A 42.0301,B 24.9431,C -1.7418,E1 25.1108,E2 404.0723} C_DIS
LIN {X 81.8988,Y 92.2209,Z 134,A 44.4991,B 24.9443,C -1.7242,E1 25.1059,E2 401.6551} C_DIS
LIN {X 79.6502,Y 94.1699,Z 134,A 46.1928,B 24.9431,C -1.7423,E1 25.1022,E2 399.925} C_DIS
LIN {X 76.5355,Y 96.7186,Z 134,A 48.0382,B 24.943,C -1.7447,E1 25.0982,E2 398.081} C_DIS
LIN {X 73.1261,Y 99.3209,Z 134,A 50.0087,B 24.9428,C -1.7472,E1 25.0938,E2 396.1118} C_DIS
LIN {X 69.1165,Y 102.1516,Z 134,A 52.2399,B 24.9427,C -1.7486,E1 25.0887,E2 393.8847} C_DIS
LIN {X 65.716,Y 104.3718,Z 134,A 54.1376,B 24.9425,C -1.7522,E1 25.0842,E2 391.9847} C_DIS
LIN {X 61.2764,Y 107.0387,Z 134,A 56.3543,B 24.9428,C -1.7465,E1 25.0789,E2 389.7883} C_DIS
LIN {X 58.3702,Y 108.6507,Z 134,A 58.104,B 24.942,C -1.7587,E1 25.0746,E2 388.0148} C_DIS
LIN {X 54.4584,Y 110.6611,Z 134,A 59.9212,B 24.9426,C -1.7504,E1 25.0701,E2 386.2223} C_DIS
LIN {X 51.7709,Y 111.9436,Z 134,A 61.4255,B 24.9421,C -1.758,E1 25.0663,E2 384.7039} C_DIS
LIN {X 48.4102,Y 113.439,Z 134,A 63.6356,B 24.9403,C -1.7843,E1 25.0604,E2 382.4367} C_DIS
LIN {X 44.6105,Y 114.9849,Z 134,A 64.9407,B 24.9421,C -1.757,E1 25.0572,E2 381.1991} C_DIS
LIN {X 41.8169,Y 116.03,Z 134,A 66.397,B 24.9418,C -1.7617,E1 25.0534,E2 379.7347} C_DIS
LIN {X 38.5259,Y 117.1648,Z 134,A 68.1762,B 24.9412,C -1.7709,E1 25.0486,E2 377.9371} C_DIS
LIN {X 34.0417,Y 118.5462,Z 134,A 70.1484,B 24.9418,C -1.7625,E1 25.0434,E2 375.9883} C_DIS
LIN {X 31.241,Y 119.3145,Z 134,A 71.5427,B 24.9416,C -1.7656,E1 25.0396,E2 374.589} C_DIS
LIN {X 26.5027,Y 120.4554,Z 134,A 73.7546,B 24.9416,C -1.7644,E1 25.0336,E2 372.3831} C_DIS
LIN {X 23.8803,Y 121.0038,Z 134,A 74.9939,B 24.9416,C -1.7647,E1 25.0302,E2 371.1446} C_DIS
LIN {X 20.9819,Y 121.5398,Z 134,A 76.9597,B 24.9397,C -1.7938,E1 25.0247,E2 369.1119} C_DIS
LIN {X 16.7641,Y 122.1922,Z 134,A 78.5521,B 24.9409,C -1.7756,E1 25.0204,E2 367.564} C_DIS
LIN {X 13.5156,Y 122.5933,Z 134,A 79.9643,B 24.9412,C -1.7707,E1 25.0165,E2 366.1644} C_DIS
LIN {X 10.1528,Y 122.9174,Z 134,A 81.4693,B 24.9414,C -1.7678,E1 25.0123,E2 364.6672} C_DIS
LIN {X 4.8408,Y 123.2408,Z 134,A 83.9095,B 24.9415,C -1.7662,E1 25.0055,E2 362.2316} C_DIS
LIN {X 0.1847,Y 123.3367,Z 134,A 86.0447,B 24.9416,C -1.7645,E1 24.9996,E2 360.1007} C_DIS
LIN {X -3.1099,Y 123.297,Z 134,A 87.6764,B 24.9414,C -1.7689,E1 24.995,E2 358.4584} C_DIS
LIN {X -7.9801,Y 123.0779,Z 134,A 90.1281,B 24.9408,C -1.7768,E1 24.9881,E2 355.9873} C_DIS
LIN {X -12.7968,Y 122.6707,Z 134,A 92.2285,B 24.9414,C -1.7689,E1 24.9823,E2 353.9045} C_DIS
LIN {X -16.5986,Y 122.215,Z 134,A 94.8166,B 24.9389,C -1.8058,E1 24.9749,E2 351.2268} C_DIS
LIN {X -22.391,Y 121.288,Z 134,A 96.6306,B 24.9419,C -1.761,E1 24.9702,E2 349.5175} C_DIS
LIN {X -28.6658,Y 119.9583,Z 134,A 99.4111,B 24.9427,C -1.7491,E1 24.9627,E2 346.7617} C_DIS
LIN {X -32.5529,Y 118.964,Z 134,A 101.6703,B 24.9416,C -1.7654,E1 24.9565,E2 344.4604} C_DIS
LIN {X -36.1533,Y 117.9177,Z 134,A 103.2644,B 24.9422,C -1.7567,E1 24.9523,E2 342.8844} C_DIS
LIN {X -39.2869,Y 116.9114,Z 134,A 104.8217,B 24.9422,C -1.7561,E1 24.9481,E2 341.3256} C_DIS
LIN {X -42.6899,Y 115.7133,Z 134,A 107.2265,B 24.9401,C -1.7876,E1 24.9416,E2 338.8411} C_DIS
LIN {X -47.4656,Y 113.836,Z 134,A 108.9462,B 24.9424,C -1.7535,E1 24.9374,E2 337.1985} C_DIS
LIN {X -50.3006,Y 112.612,Z 134,A 110.3636,B 24.9426,C -1.7506,E1 24.9338,E2 335.7846} C_DIS
LIN {X -55.6094,Y 110.0878,Z 134,A 112.8723,B 24.9435,C -1.7361,E1 24.9275,E2 333.304} C_DIS
LIN {X -58.6422,Y 108.5045,Z 134,A 114.7472,B 24.9428,C -1.7463,E1 24.9228,E2 331.3996} C_DIS
LIN {X -62.2663,Y 106.466,Z 134,A 116.6654,B 24.9431,C -1.7422,E1 24.9182,E2 329.4854} C_DIS
LIN {X -65.7578,Y 104.3454,Z 134,A 118.5206,B 24.9435,C -1.7367,E1 24.9138,E2 327.6375} C_DIS
LIN {X -68.7228,Y 102.4173,Z 134,A 120.2487,B 24.9435,C -1.7373,E1 24.9098,E2 325.9023} C_DIS
LIN {X -72.1849,Y 100.0072,Z 134,A 122.2241,B 24.9436,C -1.734,E1 24.9053,E2 323.9279} C_DIS
LIN {X -75.6492,Y 97.4128,Z 134,A 124.2308,B 24.9439,C -1.7295,E1 24.9008,E2 321.9246} C_DIS
LIN {X -78.9043,Y 94.7959,Z 134,A 126.1701,B 24.9442,C -1.7251,E1 24.8966,E2 319.9884} C_DIS
LIN {X -82.0244,Y 92.1095,Z 134,A 128.1377,B 24.9444,C -1.7232,E1 24.8925,E2 318.0177} C_DIS
LIN {X -85.2735,Y 89.1094,Z 134,A 130.1508,B 24.9448,C -1.7164,E1 24.8884,E2 316.0124} C_DIS
LIN {X -88.1035,Y 86.3124,Z 134,A 132.0125,B 24.945,C -1.7125,E1 24.8848,E2 314.1522} C_DIS
LIN {X -91.0878,Y 83.1577,Z 134,A 134.0905,B 24.9452,C -1.7101,E1 24.8808,E2 312.0708} C_DIS
LIN {X -94.0198,Y 79.8269,Z 134,A 136.1124,B 24.9457,C -1.7029,E1 24.8771,E2 310.0567} C_DIS
LIN {X -96.775,Y 76.4642,Z 134,A 138.1942,B 24.9458,C -1.7003,E1 24.8735,E2 307.9715} C_DIS
LIN {X -99.5236,Y 72.8502,Z 134,A 140.2826,B 24.9462,C -1.6936,E1 24.87,E2 305.8891} C_DIS
LIN {X -101.7702,Y 69.6771,Z 134,A 142.2342,B 24.9462,C -1.695,E1 24.8669,E2 303.9245} C_DIS
LIN {X -103.6719,Y 66.8157,Z 134,A 143.707,B 24.9468,C -1.6849,E1 24.8647,E2 302.4682} C_DIS
LIN {X -105.8646,Y 63.2831,Z 134,A 145.6573,B 24.9471,C -1.6802,E1 24.8618,E2 300.5193} C_DIS
LIN {X -108.0243,Y 59.522,Z 134,A 147.6238,B 24.9476,C -1.6721,E1 24.8591,E2 298.5617} C_DIS
LIN {X -111.2254,Y 53.2966,Z 134,A 150.7594,B 24.9485,C -1.6571,E1 24.8552,E2 295.445} C_DIS
LIN {X -112.5126,Y 50.5228,Z 134,A 152.3288,B 24.9485,C -1.6593,E1 24.8534,E2 293.8617} C_DIS
LIN {X -113.9958,Y 47.0829,Z 134,A 154.1535,B 24.9485,C -1.6577,E1 24.8514,E2 292.0309} C_DIS
LIN {X -115.5371,Y 43.1602,Z 134,A 156.0009,B 24.9492,C -1.6467,E1 24.8496,E2 290.1992} C_DIS
LIN {X -116.6904,Y 39.9401,Z 134,A 157.719,B 24.9492,C -1.6473,E1 24.848,E2 288.4698} C_DIS
LIN {X -118.0742,Y 35.6417,Z 134,A 159.8066,B 24.9496,C -1.6402,E1 24.8462,E2 286.3872} C_DIS
LIN {X -119.1815,Y 31.7399,Z 134,A 161.6034,B 24.9502,C -1.6303,E1 24.8449,E2 284.6036} C_DIS
LIN {X -119.9984,Y 28.4992,Z 134,A 163.2841,B 24.9502,C -1.6309,E1 24.8438,E2 282.9115} C_DIS
LIN {X -120.9915,Y 23.938,Z 134,A 165.5891,B 24.9502,C -1.6299,E1 24.8425,E2 280.5954} C_DIS
LIN {X -121.6387,Y 20.3892,Z 134,A 167.0794,B 24.9511,C -1.6163,E1 24.8418,E2 279.1288} C_DIS
LIN {X -122.1891,Y 16.7915,Z 134,A 169.175,B 24.9503,C -1.6286,E1 24.841,E2 276.9912} C_DIS
LIN {X -122.6216,Y 13.2526,Z 134,A 170.4517,B 24.9516,C -1.6064,E1 24.8406,E2 275.7599} C_DIS
LIN {X -122.9352,Y 9.9415,Z 134,A 171.8749,B 24.9523,C -1.596,E1 24.8402,E2 274.353} C_DIS
LIN {X -123.1339,Y 7.0725,Z 134,A 174.1786,B 24.9499,C -1.6345,E1 24.8399,E2 271.9435} C_DIS
LIN {X -123.3307,Y 1.2965,Z 134,A 175.8535,B 24.9532,C -1.5808,E1 24.8399,E2 270.3865} C_DIS
LIN {X -123.3004,Y -2.9588,Z 134,A 178.1625,B 24.9527,C -1.589,E1 24.8399,E2 268.044} C_DIS
LIN {X -123.1718,Y -6.3607,Z 134,A -179.5292,B 24.9511,C -1.6163,E1 24.8403,E2 265.657} C_DIS
LIN {X -122.7381,Y -12.1316,Z 134,A -177.0403,B 24.9521,C -1.5986,E1 24.8409,E2 263.1953} C_DIS
LIN {X -122.1773,Y -16.8739,Z 134,A -175.5578,B 24.9545,C -1.5587,E1 24.8414,E2 261.799} C_DIS
LIN {X -121.3126,Y -22.2475,Z 134,A -172.6789,B 24.954,C -1.5662,E1 24.8428,E2 258.8852} C_DIS
LIN {X -120.579,Y -25.9299,Z 134,A -171.1469,B 24.9549,C -1.5512,E1 24.8436,E2 257.3798} C_DIS
LIN {X -119.7331,Y -29.5999,Z 134,A -169.2053,B 24.9547,C -1.5542,E1 24.8449,E2 255.4197} C_DIS
LIN {X -118.7304,Y -33.3881,Z 134,A -167.5539,B 24.9555,C -1.5411,E1 24.8461,E2 253.79} C_DIS
LIN {X -117.5858,Y -37.2199,Z 134,A -165.665,B 24.9558,C -1.5368,E1 24.8477,E2 251.9004} C_DIS
LIN {X -114.3032,Y -46.3297,Z 134,A -161.2619,B 24.9568,C -1.5189,E1 24.8519,E2 247.5151} C_DIS
LIN {X -111.5673,Y -52.581,Z 134,A -158.043,B 24.9572,C -1.5118,E1 24.8555,E2 244.2955} C_DIS
LIN {X -109.5276,Y -56.708,Z 134,A -155.7726,B 24.9572,C -1.5116,E1 24.8584,E2 242.0133} C_DIS
LIN {X -105.9468,Y -63.1454,Z 134,A -152.4881,B 24.9581,C -1.496,E1 24.8629,E2 238.7488} C_DIS
LIN {X -102.9684,Y -67.8937,Z 134,A -149.9043,B 24.9585,C -1.4881,E1 24.8668,E2 236.1706} C_DIS
LIN {X -101.2972,Y -70.3629,Z 134,A -148.2622,B 24.9581,C -1.4961,E1 24.8694,E2 234.5013} C_DIS
LIN {X -99.0054,Y -73.5526,Z 134,A -146.4506,B 24.9584,C -1.491,E1 24.8723,E2 232.6933} C_DIS
LIN {X -96.4619,Y -76.858,Z 134,A -144.373,B 24.9583,C -1.4926,E1 24.876,E2 230.602} C_DIS
LIN {X -93.3268,Y -80.6361,Z 134,A -142.2113,B 24.9589,C -1.4818,E1 24.8798,E2 228.456} C_DIS
LIN {X -90.1957,Y -84.1236,Z 134,A -140.0228,B 24.9591,C -1.4774,E1 24.8839,E2 226.2684} C_DIS
LIN {X -87.1999,Y -87.226,Z 134,A -137.9532,B 24.9591,C -1.476,E1 24.888,E2 224.1932} C_DIS
LIN {X -82.8015,Y -91.411,Z 134,A -135.3981,B 24.9602,C -1.458,E1 24.8932,E2 221.6704} C_DIS
LIN {X -80.3042,Y -93.6127,Z 134,A -133.6149,B 24.9597,C -1.4658,E1 24.897,E2 219.8618} C_DIS
LIN {X -77.0959,Y -96.2725,Z 134,A -131.7622,B 24.9602,C -1.4583,E1 24.9009,E2 218.0199} C_DIS
LIN {X -73.9875,Y -98.6815,Z 134,A -129.36,B 24.9589,C -1.4816,E1 24.9064,E2 215.5536} C_DIS
LIN {X -70.4947,Y -101.2055,Z 134,A -127.9916,B 24.9607,C -1.4489,E1 24.9094,E2 214.2584} C_DIS
LIN {X -67.5175,Y -103.2161,Z 134,A -125.7285,B 24.9593,C -1.4737,E1 24.9148,E2 211.9288} C_DIS
LIN {X -64.0661,Y -105.3929,Z 134,A -124.4507,B 24.961,C -1.4421,E1 24.9177,E2 210.7222} C_DIS
LIN {X -61.3567,Y -106.9929,Z 134,A -122.8195,B 24.9607,C -1.4478,E1 24.9217,E2 209.0724} C_DIS
LIN {X -58.2487,Y -108.7159,Z 134,A -120.9042,B 24.9602,C -1.4579,E1 24.9265,E2 207.1277} C_DIS
LIN {X -54.4276,Y -110.6763,Z 134,A -119.2142,B 24.9611,C -1.4412,E1 24.9306,E2 205.473} C_DIS
LIN {X -51.5848,Y -112.0297,Z 134,A -117.1912,B 24.9598,C -1.4658,E1 24.9359,E2 203.3865} C_DIS
LIN {X -47.6359,Y -113.7649,Z 134,A -115.7082,B 24.9612,C -1.4391,E1 24.9395,E2 201.9635} C_DIS
LIN {X -44.458,Y -115.0442,Z 134,A -114.1921,B 24.9615,C -1.434,E1 24.9434,E2 200.4563} C_DIS
LIN {X -41.4473,Y -116.1633,Z 134,A -112.4876,B 24.961,C -1.4426,E1 24.948,E2 198.7279} C_DIS
LIN {X -36.9268,Y -117.6794,Z 134,A -110.4966,B 24.9617,C -1.4303,E1 24.9532,E2 196.7626} C_DIS
LIN {X -34.3166,Y -118.4657,Z 134,A -109.1793,B 24.9616,C -1.4318,E1 24.9567,E2 195.4394} C_DIS
LIN {X -29.9853,Y -119.6355,Z 134,A -107.0859,B 24.9616,C -1.431,E1 24.9624,E2 193.3449} C_DIS
LIN {X -25.9597,Y -120.5726,Z 134,A -105.118,B 24.9616,C -1.4323,E1 24.9678,E2 191.3714} C_DIS
LIN {X -20.3005,Y -121.6535,Z 134,A -102.3607,B 24.9614,C -1.4352,E1 24.9754,E2 188.6043} C_DIS
LIN {X -17.1338,Y -122.1401,Z 134,A -100.8699,B 24.9614,C -1.4349,E1 24.9795,E2 187.113} C_DIS
LIN {X -13.169,Y -122.6306,Z 134,A -99.091,B 24.9616,C -1.4309,E1 24.9844,E2 185.3423} C_DIS
LIN {X -7.8065,Y -123.0887,Z 134,A -96.5899,B 24.9616,C -1.4309,E1 24.9914,E2 182.8402} C_DIS
LIN {X -4.0617,Y -123.2706,Z 134,A -94.7358,B 24.9613,C -1.4365,E1 24.9966,E2 180.9726} C_DIS
LIN {X 0.2358,Y -123.3364,Z 134,A -92.8114,B 24.9615,C -1.4334,E1 25.0019,E2 179.0554} C_DIS
LIN {X 0.2358,Y -123.3364,Z 134,A -92.8114,B 24.9615,C -1.4334,E1 25.0019,E2 179.0554} C_DIS
Enddeposition()
LIN {X 0.8689,Y -122.3334,Z 134,A -92.8348,B 24.9614,C -1.4356,E1 25.0019,E2 179.0736} C_DIS
Startdeposition()
$VEL.CP = VEL_PRINT
LIN {X -1.9317,Y -122.3243,Z 134,A -94.6497,B 24.9627,C -1.4114,E1 24.9967,E2 180.9458} C_DIS
LIN {X -5.8886,Y -122.198,Z 134,A -96.3576,B 24.9623,C -1.4181,E1 24.9919,E2 182.6382} C_DIS
LIN {X -8.6983,Y -122.03,Z 134,A -98.0791,B 24.9633,C -1.3992,E1 24.987,E2 184.4052} C_DIS
LIN {X -13.4112,Y -121.6025,Z 134,A -100.0905,B 24.9628,C -1.409,E1 24.9815,E2 186.3945} C_DIS
LIN {X -17.7592,Y -121.0444,Z 134,A -102.0187,B 24.9625,C -1.4152,E1 24.9762,E2 188.3094} C_DIS
LIN {X -24.126,Y -119.9371,Z 134,A -105.6514,B 24.9639,C -1.3882,E1 24.966,E2 192.0099} C_DIS
LIN {X -28.279,Y -119.0267,Z 134,A -107.3166,B 24.9631,C -1.4043,E1 24.9616,E2 193.6392} C_DIS
LIN {X -32.3831,Y -117.9769,Z 134,A -109.1122,B 24.9625,C -1.4142,E1 24.9568,E2 195.414} C_DIS
LIN {X -35.3921,Y -117.1087,Z 134,A -110.677,B 24.9627,C -1.4107,E1 24.9526,E2 196.9896} C_DIS
LIN {X -40.2158,Y -115.5403,Z 134,A -112.972,B 24.9624,C -1.4164,E1 24.9465,E2 199.2755} C_DIS
LIN {X -44.0881,Y -114.119,Z 134,A -114.8146,B 24.9621,C -1.4223,E1 24.9418,E2 201.1079} C_DIS
LIN {X -51.4869,Y -110.9773,Z 134,A -118.5109,B 24.9617,C -1.4294,E1 24.9323,E2 204.7958} C_DIS
LIN {X -56.477,Y -108.5236,Z 134,A -121.2369,B 24.9618,C -1.4271,E1 24.9255,E2 207.5346} C_DIS
LIN {X -59.8534,Y -106.6999,Z 134,A -123.1001,B 24.9618,C -1.4266,E1 24.9209,E2 209.4043} C_DIS
LIN {X -63.1978,Y -104.7537,Z 134,A -124.6431,B 24.9611,C -1.4415,E1 24.9172,E2 210.9167} C_DIS
LIN {X -67.5323,Y -102.0135,Z 134,A -127.1056,B 24.9611,C -1.4424,E1 24.9114,E2 213.3848} C_DIS
LIN {X -72.4445,Y -98.5853,Z 134,A -130.1174,B 24.9613,C -1.4378,E1 24.9045,E2 216.4178} C_DIS
LIN {X -75.5694,Y -96.2109,Z 134,A -131.9585,B 24.9611,C -1.441,E1 24.9004,E2 218.258} C_DIS
LIN {X -78.5318,Y -93.8086,Z 134,A -133.8503,B 24.9611,C -1.4397,E1 24.8963,E2 220.1601} C_DIS
LIN {X -81.8947,Y -90.8882,Z 134,A -135.9662,B 24.9611,C -1.4426,E1 24.8919,E2 222.2776} C_DIS
LIN {X -86.1984,Y -86.8166,Z 134,A -138.7197,B 24.9606,C -1.4494,E1 24.8864,E2 225.0264} C_DIS
LIN {X -89.2602,Y -83.6663,Z 134,A -140.6154,B 24.96,C -1.4611,E1 24.8827,E2 226.9024} C_DIS
LIN {X -91.3837,Y -81.3415,Z 134,A -142.2944,B 24.9603,C -1.4554,E1 24.8796,E2 228.6024} C_DIS
LIN {X -94.1117,Y -78.1685,Z 134,A -144.1127,B 24.9597,C -1.4663,E1 24.8763,E2 230.4031} C_DIS
LIN {X -96.5677,Y -75.1133,Z 134,A -146.0207,B 24.9597,C -1.4675,E1 24.873,E2 232.3172} C_DIS
LIN {X -98.6953,Y -72.2949,Z 134,A -147.7674,B 24.9597,C -1.4675,E1 24.8701,E2 234.0721} C_DIS
LIN {X -101.1734,Y -68.7843,Z 134,A -149.6322,B 24.959,C -1.4792,E1 24.8671,E2 235.9183} C_DIS
LIN {X -104.0789,Y -64.3041,Z 134,A -152.3256,B 24.9591,C -1.4774,E1 24.8631,E2 238.6298} C_DIS
LIN {X -107.6001,Y -58.2206,Z 134,A -155.6293,B 24.9586,C -1.4859,E1 24.8585,E2 241.9306} C_DIS
LIN {X -109.5569,Y -54.4448,Z 134,A -157.4839,B 24.958,C -1.4975,E1 24.8562,E2 243.7674} C_DIS
LIN {X -110.6425,Y -52.2056,Z 134,A -159.2581,B 24.9593,C -1.4744,E1 24.854,E2 245.6062} C_DIS
LIN {X -112.4208,Y -48.2547,Z 134,A -160.7778,B 24.9577,C -1.5024,E1 24.8524,E2 247.0677} C_DIS
LIN {X -113.9413,Y -44.5453,Z 134,A -163.6285,B 24.9597,C -1.4661,E1 24.8494,E2 250.0208} C_DIS
LIN {X -116.1303,Y -38.4791,Z 134,A -165.6727,B 24.9569,C -1.5171,E1 24.8476,E2 251.9551} C_DIS
LIN {X -117.3424,Y -34.6078,Z 134,A -167.5973,B 24.9566,C -1.5219,E1 24.846,E2 253.8794} C_DIS
LIN {X -118.43,Y -30.6854,Z 134,A -169.5076,B 24.9563,C -1.5276,E1 24.8447,E2 255.7872} C_DIS
LIN {X -119.2502,Y -27.3181,Z 134,A -171.1288,B 24.956,C -1.5328,E1 24.8436,E2 257.4056} C_DIS
LIN {X -119.8613,Y -24.4985,Z 134,A -172.9322,B 24.9569,C -1.5176,E1 24.8426,E2 259.2557} C_DIS
LIN {X -120.5798,Y -20.6818,Z 134,A -174.4005,B 24.9557,C -1.5384,E1 24.8419,E2 260.6832} C_DIS
LIN {X -121.1359,Y -17.1188,Z 134,A -175.9612,B 24.955,C -1.5494,E1 24.8412,E2 262.227} C_DIS
LIN {X -121.6998,Y -12.5073,Z 134,A -178.6873,B 24.956,C -1.5328,E1 24.8404,E2 265.009} C_DIS
LIN {X -122.0349,Y -8.6319,Z 134,A 179.8543,B 24.9547,C -1.5543,E1 24.8401,E2 266.425} C_DIS
LIN {X -122.2695,Y -4.1786,Z 134,A 177.2805,B 24.9555,C -1.5403,E1 24.8398,E2 269.0476} C_DIS
LIN {X -122.3411,Y 0.2447,Z 134,A 175.877,B 24.9535,C -1.5757,E1 24.8398,E2 270.3752} C_DIS
LIN {X -122.162,Y 6.6038,Z 134,A 172.826,B 24.9531,C -1.5823,E1 24.8401,E2 273.4287} C_DIS
LIN {X -121.7237,Y 12.2714,Z 134,A 169.9016,B 24.9532,C -1.5798,E1 24.8408,E2 276.3767} C_DIS
LIN {X -121.2628,Y 16.1974,Z 134,A 168.2613,B 24.9523,C -1.5949,E1 24.8413,E2 277.9908} C_DIS
LIN {X -120.7987,Y 19.3653,Z 134,A 166.7251,B 24.9521,C -1.5982,E1 24.842,E2 279.5283} C_DIS
LIN {X -120.2611,Y 22.4597,Z 134,A 164.9134,B 24.9527,C -1.5884,E1 24.8429,E2 281.374} C_DIS
LIN {X -119.2362,Y 27.3796,Z 134,A 162.8428,B 24.9515,C -1.6082,E1 24.8441,E2 283.4097} C_DIS
LIN {X -118.32,Y 31.1036,Z 134,A 160.9648,B 24.9515,C -1.6104,E1 24.8454,E2 285.2932} C_DIS
LIN {X -117.3333,Y 34.6388,Z 134,A 159.3317,B 24.9508,C -1.6196,E1 24.8467,E2 286.9139} C_DIS
LIN {X -116.0053,Y 38.8544,Z 134,A 157.2263,B 24.9505,C -1.6247,E1 24.8485,E2 289.0193} C_DIS
LIN {X -114.6332,Y 42.7331,Z 134,A 155.3345,B 24.9501,C -1.6323,E1 24.8503,E2 290.9038} C_DIS
LIN {X -113.4554,Y 45.7682,Z 134,A 153.783,B 24.9499,C -1.6359,E1 24.8518,E2 292.4554} C_DIS
LIN {X -112.0692,Y 49.0679,Z 134,A 152.1007,B 24.9496,C -1.6408,E1 24.8537,E2 294.1353} C_DIS
LIN {X -110.5091,Y 52.4848,Z 134,A 150.5455,B 24.9487,C -1.655,E1 24.8555,E2 295.6652} C_DIS
LIN {X -108.7029,Y 56.1314,Z 134,A 148.4112,B 24.9489,C -1.6508,E1 24.8582,E2 297.8208} C_DIS
LIN {X -106.3015,Y 60.558,Z 134,A 145.927,B 24.9489,C -1.6524,E1 24.8615,E2 300.3144} C_DIS
LIN {X -104.1621,Y 64.1685,Z 134,A 143.8116,B 24.9489,C -1.6516,E1 24.8646,E2 302.4425} C_DIS
LIN {X -101.4741,Y 68.3401,Z 134,A 141.6738,B 24.948,C -1.6663,E1 24.8679,E2 304.5561} C_DIS
LIN {X -99.1606,Y 71.6553,Z 134,A 139.695,B 24.9479,C -1.6679,E1 24.8711,E2 306.5408} C_DIS
LIN {X -96.5099,Y 75.1878,Z 134,A 137.6562,B 24.9474,C -1.6748,E1 24.8745,E2 308.5729} C_DIS
LIN {X -93.932,Y 78.3847,Z 134,A 135.6587,B 24.9474,C -1.6767,E1 24.8781,E2 310.5751} C_DIS
LIN {X -91.0166,Y 81.7514,Z 134,A 133.5934,B 24.9469,C -1.6829,E1 24.8819,E2 312.6347} C_DIS
LIN {X -88.1115,Y 84.8748,Z 134,A 131.5553,B 24.9467,C -1.6862,E1 24.8858,E2 314.674} C_DIS
LIN {X -84.9951,Y 87.9951,Z 134,A 129.5253,B 24.9463,C -1.6928,E1 24.8898,E2 316.6968} C_DIS
LIN {X -81.9113,Y 90.8734,Z 134,A 127.4945,B 24.9462,C -1.695,E1 24.894,E2 318.7305} C_DIS
LIN {X -78.7221,Y 93.6489,Z 134,A 125.5346,B 24.9458,C -1.7004,E1 24.8981,E2 320.6852} C_DIS
LIN {X -75.3465,Y 96.386,Z 134,A 123.4734,B 24.9456,C -1.7038,E1 24.9026,E2 322.7461} C_DIS
LIN {X -71.977,Y 98.9275,Z 134,A 121.4852,B 24.9454,C -1.7074,E1 24.9071,E2 324.7327} C_DIS
LIN {X -68.2744,Y 101.5186,Z 134,A 119.3342,B 24.9452,C -1.7102,E1 24.912,E2 326.8843} C_DIS
LIN {X -64.8725,Y 103.7252,Z 134,A 117.45,B 24.9449,C -1.7145,E1 24.9165,E2 328.7643} C_DIS
LIN {X -61.0864,Y 105.999,Z 134,A 115.423,B 24.9446,C -1.7201,E1 24.9213,E2 330.7842} C_DIS
LIN {X -57.671,Y 107.8954,Z 134,A 113.6616,B 24.9441,C -1.7263,E1 24.9256,E2 332.5358} C_DIS
LIN {X -55.488,Y 109.0317,Z 134,A 112.278,B 24.9447,C -1.718,E1 24.9291,E2 333.9428} C_DIS
LIN {X -51.7026,Y 110.8776,Z 134,A 110.4864,B 24.944,C -1.7292,E1 24.9336,E2 335.7125} C_DIS
LIN {X -48.5254,Y 112.3037,Z 134,A 108.8887,B 24.9437,C -1.7331,E1 24.9376,E2 337.3047} C_DIS
LIN {X -41.4023,Y 115.1204,Z 134,A 105.2282,B 24.9437,C -1.7347,E1 24.9472,E2 340.9692} C_DIS
LIN {X -37.446,Y 116.4676,Z 134,A 103.3474,B 24.9432,C -1.7405,E1 24.9521,E2 342.8396} C_DIS
LIN {X -34.9574,Y 117.24,Z 134,A 101.8488,B 24.944,C -1.7294,E1 24.9562,E2 344.3673} C_DIS
LIN {X -30.6742,Y 118.4328,Z 134,A 100.0562,B 24.943,C -1.7446,E1 24.961,E2 346.1265} C_DIS
LIN {X -27.9188,Y 119.1129,Z 134,A 98.1239,B 24.9446,C -1.7187,E1 24.9664,E2 348.1229} C_DIS
LIN {X -23.7582,Y 120.0119,Z 134,A 96.7435,B 24.9427,C -1.748,E1 24.97,E2 349.4352} C_DIS
LIN {X -16.5045,Y 121.2225,Z 134,A 93.1581,B 24.943,C -1.744,E1 24.9799,E2 353.0334} C_DIS
LIN {X -10.2836,Y 121.9065,Z 134,A 90.4138,B 24.9423,C -1.7541,E1 24.9875,E2 355.7554} C_DIS
LIN {X -4.5487,Y 122.2551,Z 134,A 87.4973,B 24.943,C -1.7447,E1 24.9957,E2 358.6949} C_DIS
LIN {X -1.5518,Y 122.3307,Z 134,A 85.5898,B 24.9444,C -1.722,E1 25.0012,E2 360.6563} C_DIS
LIN {X 2.9621,Y 122.3044,Z 134,A 84.2462,B 24.9421,C -1.7576,E1 25.0047,E2 361.9153} C_DIS
LIN {X 9.0118,Y 122.0071,Z 134,A 81.2523,B 24.9426,C -1.7504,E1 25.0131,E2 364.9253} C_DIS
LIN {X 14.9604,Y 121.4221,Z 134,A 78.3059,B 24.9431,C -1.7431,E1 25.0213,E2 367.887} C_DIS
LIN {X 19.7743,Y 120.7312,Z 134,A 76.22,B 24.9425,C -1.7514,E1 25.027,E2 369.9513} C_DIS
LIN {X 25.0359,Y 119.7516,Z 134,A 73.4096,B 24.9435,C -1.7361,E1 25.0348,E2 372.7947} C_DIS
LIN {X 29.36,Y 118.7661,Z 134,A 71.5858,B 24.9428,C -1.7467,E1 25.0396,E2 374.5905} C_DIS
LIN {X 32.4937,Y 117.946,Z 134,A 69.9171,B 24.9433,C -1.7386,E1 25.0442,E2 376.2758} C_DIS
LIN {X 37.7185,Y 116.3806,Z 134,A 67.3928,B 24.9433,C -1.7381,E1 25.0509,E2 378.7969} C_DIS
LIN {X 41.3839,Y 115.1271,Z 134,A 65.7069,B 24.9431,C -1.7425,E1 25.0553,E2 380.4689} C_DIS
LIN {X 46.5182,Y 113.1516,Z 134,A 62.8496,B 24.9441,C -1.7266,E1 25.0628,E2 383.3575} C_DIS
LIN {X 50.2601,Y 111.5387,Z 134,A 61.22,B 24.9434,C -1.7376,E1 25.0669,E2 384.9571} C_DIS
LIN {X 54.2821,Y 109.6372,Z 134,A 59.1936,B 24.9434,C -1.7378,E1 25.072,E2 386.9778} C_DIS
LIN {X 57.4949,Y 107.9891,Z 134,A 57.4239,B 24.9438,C -1.7317,E1 25.0764,E2 388.7568} C_DIS
LIN {X 61.0374,Y 106.0274,Z 134,A 55.426,B 24.9443,C -1.7241,E1 25.0813,E2 390.7667} C_DIS
LIN {X 65.1952,Y 103.5224,Z 134,A 53.3862,B 24.9438,C -1.7318,E1 25.0861,E2 392.7819} C_DIS
LIN {X 67.963,Y 101.7265,Z 134,A 51.647,B 24.9446,C -1.72,E1 25.0902,E2 394.5433} C_DIS
LIN {X 71.2846,Y 99.4274,Z 134,A 49.8049,B 24.9446,C -1.7191,E1 25.0944,E2 396.3812} C_DIS
LIN {X 74.5054,Y 97.0375,Z 134,A 47.9249,B 24.9448,C -1.7156,E1 25.0986,E2 398.2626} C_DIS
LIN {X 76.8861,Y 95.1621,Z 134,A 46.5648,B 24.9448,C -1.7158,E1 25.1015,E2 399.6172} C_DIS
LIN {X 79.8606,Y 92.6799,Z 134,A 44.7575,B 24.945,C -1.7126,E1 25.1054,E2 401.4251} C_DIS
LIN {X 82.4184,Y 90.4133,Z 134,A 42.699,B 24.9467,C -1.6871,E1 25.1098,E2 403.5354} C_DIS
LIN {X 85.3964,Y 87.6063,Z 134,A 41.1795,B 24.9457,C -1.7023,E1 25.1127,E2 405.0128} C_DIS
LIN {X 88.3822,Y 84.5924,Z 134,A 39.1616,B 24.9461,C -1.6964,E1 25.1166,E2 407.0359} C_DIS
LIN {X 91.4444,Y 81.273,Z 134,A 37.1041,B 24.9462,C -1.6943,E1 25.1205,E2 409.0892} C_DIS
LIN {X 93.5641,Y 78.8232,Z 134,A 35.2962,B 24.9473,C -1.6765,E1 25.1238,E2 410.9308} C_DIS
LIN {X 95.8492,Y 76.0279,Z 134,A 33.96,B 24.9465,C -1.6897,E1 25.1261,E2 412.2296} C_DIS
LIN {X 98.3932,Y 72.7061,Z 134,A 32.1257,B 24.9465,C -1.691,E1 25.1291,E2 414.0521} C_DIS
LIN {X 100.273,Y 70.0891,Z 134,A 30.1965,B 24.948,C -1.6665,E1 25.1323,E2 416.0297} C_DIS
LIN {X 102.2359,Y 67.1945,Z 134,A 28.8806,B 24.9472,C -1.678,E1 25.1343,E2 417.3118} C_DIS
LIN {X 104.4719,Y 63.6634,Z 134,A 26.8744,B 24.9477,C -1.6704,E1 25.1373,E2 419.326} C_DIS
LIN {X 106.6819,Y 59.8854,Z 134,A 24.8624,B 24.9479,C -1.6666,E1 25.1401,E2 421.3364} C_DIS
LIN {X 108.1971,Y 57.0988,Z 134,A 23.4491,B 24.9479,C -1.6661,E1 25.1419,E2 422.7436} C_DIS
LIN {X 110.7416,Y 51.9966,Z 134,A 20.7195,B 24.9486,C -1.6555,E1 25.1453,E2 425.4835} C_DIS
LIN {X 112.2233,Y 48.7114,Z 134,A 19.1587,B 24.9486,C -1.6569,E1 25.147,E2 427.0326} C_DIS
LIN {X 113.28,Y 46.2032,Z 134,A 17.8924,B 24.9488,C -1.6535,E1 25.1484,E2 428.2997} C_DIS
LIN {X 114.4891,Y 43.1179,Z 134,A 16.3114,B 24.9491,C -1.6475,E1 25.15,E2 429.8863} C_DIS
LIN {X 115.7942,Y 39.4837,Z 134,A 14.4372,B 24.9497,C -1.6387,E1 25.1517,E2 431.7706} C_DIS
LIN {X 116.6933,Y 36.7396,Z 134,A 12.7464,B 24.951,C -1.6177,E1 25.1532,E2 433.5012} C_DIS
LIN {X 117.7723,Y 33.1149,Z 134,A 11.4519,B 24.9498,C -1.636,E1 25.1541,E2 434.7454} C_DIS
LIN {X 118.6201,Y 29.9363,Z 134,A 9.9001,B 24.9502,C -1.6306,E1 25.1552,E2 436.3009} C_DIS
LIN {X 119.3646,Y 26.8173,Z 134,A 8.3503,B 24.9506,C -1.6235,E1 25.1562,E2 437.8585} C_DIS
LIN {X 120.7565,Y 19.6226,Z 134,A 4.9063,B 24.9513,C -1.6119,E1 25.1579,E2 441.3096} C_DIS
LIN {X 121.7045,Y 12.4635,Z 134,A 1.1367,B 24.9531,C -1.5816,E1 25.1592,E2 445.1282} C_DIS
LIN {X 122.0533,Y 8.3791,Z 134,A -0.3405,B 24.9522,C -1.5975,E1 25.1595,E2 446.5593} C_DIS
LIN {X 122.23,Y 5.1937,Z 134,A -1.9063,B 24.9527,C -1.589,E1 25.1597,E2 448.1358} C_DIS
LIN {X 122.3398,Y 0.4983,Z 134,A -3.9356,B 24.9527,C -1.5903,E1 25.1597,E2 450.1499} C_DIS
LIN {X 122.3016,Y -3.0658,Z 134,A -5.6121,B 24.953,C -1.5845,E1 25.1597,E2 451.8301} C_DIS
LIN {X 122.1547,Y -6.7495,Z 134,A -7.4136,B 24.9535,C -1.575,E1 25.1595,E2 453.6432} C_DIS
LIN {X 121.8302,Y -11.1634,Z 134,A -9.4827,B 24.9539,C -1.5684,E1 25.159,E2 455.7157} C_DIS
LIN {X 121.0085,Y -18.0098,Z 134,A -12.6075,B 24.9542,C -1.563,E1 25.1579,E2 458.8347} C_DIS
LIN {X 119.6678,Y -25.4296,Z 134,A -16.7489,B 24.9567,C -1.5211,E1 25.1556,E2 463.0508} C_DIS
LIN {X 118.5576,Y -30.1825,Z 134,A -18.3732,B 24.9552,C -1.5467,E1 25.1546,E2 464.6054} C_DIS
LIN {X 117.643,Y -33.5772,Z 134,A -20.8295,B 24.9578,C -1.501,E1 25.1527,E2 467.1553} C_DIS
LIN {X 115.9506,Y -39.0188,Z 134,A -22.6113,B 24.9558,C -1.5367,E1 25.1512,E2 468.8429} C_DIS
LIN {X 114.6737,Y -42.6249,Z 134,A -24.4244,B 24.9561,C -1.53,E1 25.1494,E2 470.6617} C_DIS
LIN {X 113.4795,Y -45.7083,Z 134,A -27.016,B 24.9593,C -1.4733,E1 25.1466,E2 473.3726} C_DIS
LIN {X 110.7416,Y -51.9965,Z 134,A -29.1012,B 24.9568,C -1.5193,E1 25.1443,E2 475.3381} C_DIS
LIN {X 106.6623,Y -59.9203,Z 134,A -33.3947,B 24.9578,C -1.5007,E1 25.1387,E2 479.6527} C_DIS
LIN {X 104.4819,Y -63.6472,Z 134,A -35.4237,B 24.9582,C -1.4944,E1 25.1358,E2 481.6861} C_DIS
LIN {X 102.0819,Y -67.4284,Z 134,A -37.3974,B 24.9582,C -1.4945,E1 25.1328,E2 483.6497} C_DIS
LIN {X 100.0214,Y -70.4486,Z 134,A -39.1431,B 24.9585,C -1.488,E1 25.13,E2 485.4021} C_DIS
LIN {X 95.0079,Y -77.0773,Z 134,A -43.0759,B 24.9592,C -1.4753,E1 25.1233,E2 489.3462} C_DIS
LIN {X 92.4118,Y -80.1715,Z 134,A -45.3284,B 24.9605,C -1.4525,E1 25.1192,E2 491.6424} C_DIS
LIN {X 89.7203,Y -83.1722,Z 134,A -46.7122,B 24.9594,C -1.4725,E1 25.1166,E2 492.9728} C_DIS
LIN {X 85.8683,Y -87.1435,Z 134,A -49.3677,B 24.9599,C -1.4629,E1 25.1114,E2 495.6398} C_DIS
LIN {X 80.9876,Y -91.6967,Z 134,A -52.346,B 24.9599,C -1.4627,E1 25.1053,E2 498.6065} C_DIS
LIN {X 77.6562,Y -94.5351,Z 134,A -54.549,B 24.9606,C -1.4504,E1 25.1006,E2 500.8299} C_DIS
LIN {X 74.8161,Y -96.798,Z 134,A -56.5739,B 24.9617,C -1.4308,E1 25.096,E2 502.8937} C_DIS
LIN {X 71.7873,Y -99.065,Z 134,A -58.0719,B 24.9611,C -1.4404,E1 25.0927,E2 504.3636} C_DIS
LIN {X 67.7968,Y -101.8376,Z 134,A -60.1512,B 24.9609,C -1.4454,E1 25.0879,E2 506.4241} C_DIS
LIN {X 65.0325,Y -103.6251,Z 134,A -61.7045,B 24.9611,C -1.4418,E1 25.0843,E2 507.9809} C_DIS
LIN {X 59.0069,Y -107.1707,Z 134,A -65.0296,B 24.9615,C -1.4333,E1 25.0762,E2 511.3161} C_DIS
LIN {X 55.8331,Y -108.856,Z 134,A -66.6034,B 24.9614,C -1.4357,E1 25.0723,E2 512.8797} C_DIS
LIN {X 52.7103,Y -110.4014,Z 134,A -68.8175,B 24.963,C -1.4049,E1 25.0666,E2 515.161} C_DIS
LIN {X 48.7597,Y -112.2024,Z 134,A -70.2822,B 24.9617,C -1.4292,E1 25.063,E2 516.5645} C_DIS
LIN {X 45.1938,Y -113.6869,Z 134,A -72.2696,B 24.9623,C -1.4179,E1 25.0578,E2 518.574} C_DIS
LIN {X 40.8129,Y -115.3329,Z 134,A -74.3978,B 24.9623,C -1.418,E1 25.0522,E2 520.6976} C_DIS
LIN {X 37.1423,Y -116.5647,Z 134,A -76.1244,B 24.9623,C -1.42,E1 25.0477,E2 522.4162} C_DIS
LIN {X 33.5859,Y -117.6404,Z 134,A -78.8946,B 24.9649,C -1.3689,E1 25.04,E2 525.3027} C_DIS
LIN {X 27.0668,Y -119.3076,Z 134,A -80.7741,B 24.9619,C -1.4263,E1 25.0352,E2 527.0436} C_DIS
LIN {X 24.6801,Y -119.8243,Z 134,A -82.8638,B 24.9643,C -1.3802,E1 25.0292,E2 529.2398} C_DIS
LIN {X 19.4154,Y -120.7909,Z 134,A -84.5533,B 24.9624,C -1.417,E1 25.0248,E2 530.8405} C_DIS
LIN {X 13.3801,Y -121.6059,Z 134,A -87.4978,B 24.9627,C -1.4108,E1 25.0166,E2 533.7975} C_DIS
LIN {X 10.1431,Y -121.9183,Z 134,A -89.3034,B 24.9635,C -1.3966,E1 25.0115,E2 535.6356} C_DIS
LIN {X 6.8672,Y -122.1476,Z 134,A -90.7016,B 24.9632,C -1.4025,E1 25.0076,E2 537.0192} C_DIS
LIN {X 2.1371,Y -122.3209,Z 134,A -92.7712,B 24.9628,C -1.4088,E1 25.0019,E2 539.0736} C_DIS
LIN {X 2.1371,Y -122.3209,Z 134,A -92.7712,B 24.9628,C -1.4088,E1 25.0019,E2 539.0736} C_DIS
Enddeposition()
LIN {X 0.8558,Y -121.3391,Z 134,A -92.6969,B 24.9602,C -1.458,E1 25.0024,E2 538.8827} C_DIS
Startdeposition()
$VEL.CP = VEL_PRINT
LIN {X 3.9313,Y -121.2808,Z 134,A -91.2677,B 24.9602,C -1.4573,E1 25.0064,E2 537.4554} C_DIS
LIN {X 12.1387,Y -120.7357,Z 134,A -87.5079,B 24.9604,C -1.4531,E1 25.0169,E2 533.7074} C_DIS
LIN {X 19.5105,Y -119.7651,Z 134,A -83.8473,B 24.9599,C -1.4626,E1 25.0271,E2 530.0274} C_DIS
LIN {X 25.582,Y -118.6157,Z 134,A -81.0216,B 24.96,C -1.4606,E1 25.0348,E2 527.2097} C_DIS
LIN {X 28.6931,Y -117.902,Z 134,A -79.3459,B 24.9595,C -1.4702,E1 25.0394,E2 525.5136} C_DIS
LIN {X 34.9661,Y -116.1972,Z 134,A -76.4516,B 24.9598,C -1.4651,E1 25.0471,E2 522.6362} C_DIS
LIN {X 38.7424,Y -114.9926,Z 134,A -74.516,B 24.9595,C -1.4705,E1 25.0523,E2 520.6915} C_DIS
LIN {X 42.043,Y -113.8278,Z 134,A -72.1011,B 24.9573,C -1.51,E1 25.0588,E2 518.1882} C_DIS
LIN {X 46.7216,Y -111.9873,Z 134,A -70.4718,B 24.9591,C -1.4769,E1 25.0628,E2 516.6409} C_DIS
LIN {X 52.3723,Y -109.4587,Z 134,A -67.18,B 24.9579,C -1.4996,E1 25.0713,E2 513.3038} C_DIS
LIN {X 55.4638,Y -107.926,Z 134,A -65.9342,B 24.9588,C -1.4835,E1 25.0743,E2 512.0994} C_DIS
LIN {X 58.8874,Y -106.098,Z 134,A -63.8876,B 24.958,C -1.4973,E1 25.0794,E2 510.0263} C_DIS
LIN {X 61.9927,Y -104.3141,Z 134,A -62.4865,B 24.9586,C -1.4861,E1 25.0827,E2 508.6557} C_DIS
LIN {X 64.0661,Y -103.0536,Z 134,A -61.3943,B 24.9586,C -1.4857,E1 25.0853,E2 507.5679} C_DIS
LIN {X 66.6698,Y -101.3886,Z 134,A -59.8563,B 24.9583,C -1.4925,E1 25.0889,E2 506.0191} C_DIS
LIN {X 68.8731,Y -99.9052,Z 134,A -58.452,B 24.9577,C -1.5024,E1 25.0922,E2 504.596} C_DIS
LIN {X 71.7374,Y -97.8685,Z 134,A -56.8684,B 24.9577,C -1.5022,E1 25.0957,E2 503.0185} C_DIS
LIN {X 74.8013,Y -95.5474,Z 134,A -55.0525,B 24.9575,C -1.5062,E1 25.0998,E2 501.1998} C_DIS
LIN {X 77.7946,Y -93.1266,Z 134,A -53.1903,B 24.9571,C -1.5125,E1 25.1038,E2 499.3298} C_DIS
LIN {X 81.448,Y -89.9485,Z 134,A -50.7953,B 24.9565,C -1.5233,E1 25.1088,E2 496.9189} C_DIS
LIN {X 84.7769,Y -86.8185,Z 134,A -48.7708,B 24.9566,C -1.5219,E1 25.1129,E2 494.906} C_DIS
LIN {X 87.7465,Y -83.8155,Z 134,A -46.5696,B 24.9557,C -1.5373,E1 25.1172,E2 492.678} C_DIS
LIN {X 89.9335,Y -81.4645,Z 134,A -45.3131,B 24.9562,C -1.5282,E1 25.1195,E2 491.4485} C_DIS
LIN {X 91.9563,Y -79.1741,Z 134,A -43.8691,B 24.956,C -1.532,E1 25.1222,E2 490.002} C_DIS
LIN {X 94.5941,Y -76.0032,Z 134,A -41.952,B 24.9558,C -1.5357,E1 25.1255,E2 488.0851} C_DIS
LIN {X 97.6707,Y -72.0068,Z 134,A -39.9132,B 24.9564,C -1.5252,E1 25.1289,E2 486.0809} C_DIS
LIN {X 99.2082,Y -69.8731,Z 134,A -38.3223,B 24.9552,C -1.5461,E1 25.1316,E2 484.4484} C_DIS
LIN {X 101.2342,Y -66.9043,Z 134,A -36.774,B 24.9554,C -1.5435,E1 25.134,E2 482.9139} C_DIS
LIN {X 103.1866,Y -63.8523,Z 134,A -34.9235,B 24.9547,C -1.5554,E1 25.1367,E2 481.0445} C_DIS
LIN {X 105.3262,Y -60.2571,Z 134,A -33.1089,B 24.9548,C -1.5532,E1 25.1393,E2 479.2446} C_DIS
LIN {X 107.9559,Y -55.4051,Z 134,A -30.5375,B 24.9544,C -1.5593,E1 25.1427,E2 476.6724} C_DIS
LIN {X 109.5221,Y -52.2395,Z 134,A -28.789,B 24.9539,C -1.5684,E1 25.1448,E2 474.9117} C_DIS
LIN {X 111.239,Y -48.4774,Z 134,A -26.4692,B 24.9525,C -1.593,E1 25.1475,E2 472.5465} C_DIS
LIN {X 112.6195,Y -45.1769,Z 134,A -25.4055,B 24.954,C -1.5667,E1 25.1485,E2 471.5508} C_DIS
LIN {X 113.5938,Y -42.6678,Z 134,A -23.9244,B 24.9532,C -1.5813,E1 25.15,E2 470.0435} C_DIS
LIN {X 114.8727,Y -39.1001,Z 134,A -22.1965,B 24.953,C -1.5838,E1 25.1516,E2 468.3194} C_DIS
LIN {X 116.2056,Y -34.9384,Z 134,A -19.9245,B 24.952,C -1.6009,E1 25.1535,E2 466.0199} C_DIS
LIN {X 117.2683,Y -31.1808,Z 134,A -18.2475,B 24.9521,C -1.5985,E1 25.1548,E2 464.3584} C_DIS
LIN {X 117.9907,Y -28.325,Z 134,A -16.7213,B 24.9514,C -1.6098,E1 25.1558,E2 462.8143} C_DIS
LIN {X 118.7038,Y -25.1739,Z 134,A -15.2673,B 24.9514,C -1.6111,E1 25.1566,E2 461.3656} C_DIS
LIN {X 119.8429,Y -19.0272,Z 134,A -12.6041,B 24.9517,C -1.6062,E1 25.1579,E2 458.7296} C_DIS
LIN {X 120.7128,Y -12.3673,Z 134,A -9.1018,B 24.95,C -1.6332,E1 25.1591,E2 455.1843} C_DIS
LIN {X 121.0847,Y -7.9294,Z 134,A -7.1351,B 24.95,C -1.6332,E1 25.1595,E2 453.2291} C_DIS
LIN {X 121.2773,Y -4.0545,Z 134,A -5.458,B 24.9501,C -1.6315,E1 25.1597,E2 451.5662} C_DIS
LIN {X 121.3324,Y -1.6604,Z 134,A -4.1928,B 24.9495,C -1.642,E1 25.1597,E2 450.2838} C_DIS
LIN {X 121.3187,Y 2.4828,Z 134,A -2.0412,B 24.9485,C -1.6583,E1 25.1597,E2 448.1067} C_DIS
LIN {X 121.12,Y 7.3569,Z 134,A 0.763,B 24.9464,C -1.6913,E1 25.1592,E2 445.2414} C_DIS
LIN {X 120.6653,Y 12.8087,Z 134,A 3.1938,B 24.9464,C -1.6919,E1 25.1585,E2 442.8235} C_DIS
LIN {X 120.0551,Y 17.6388,Z 134,A 4.7215,B 24.9483,C -1.6602,E1 25.158,E2 441.3794} C_DIS
LIN {X 118.4189,Y 26.4835,Z 134,A 9.0048,B 24.9474,C -1.6754,E1 25.1557,E2 437.0853} C_DIS
LIN {X 117.6113,Y 29.861,Z 134,A 10.7016,B 24.9469,C -1.6835,E1 25.1546,E2 435.3794} C_DIS
LIN {X 116.8262,Y 32.7985,Z 134,A 12.1082,B 24.9467,C -1.6864,E1 25.1535,E2 433.9738} C_DIS
Enddeposition()
END
